LIN {X 0,Y 273.88,Z 288.831,A -85,B 0,C 180,E1 -19129.181,E2 -19129.181} C_VEL
LIN {X 0,Y 275.727,Z 293.143,A -85,B 0,C 180,E1 -19129.643,E2 -19129.643} C_VEL
LIN {X 0,Y 275.975,Z 296.307,A -85,B 0,C 180,E1 -19129.792,E2 -19129.792} C_VEL
LIN {X 0,Y 270.634,Z 402.684,A -85,B 0,C 180,E1 -19132.569,E2 -19132.569} C_VEL
LIN {X 0,Y 269.012,Z 418.51,A -85,B 0,C 180,E1 -19133.244,E2 -19133.244} C_VEL
LIN {X 0,Y 266.872,Z 432.935,A -85,B 0,C 180,E1 -19134.131,E2 -19134.131} C_VEL
LIN {X 0,Y 264.208,Z 447.475,A -85,B 0,C 180,E1 -19135.35,E2 -19135.35} C_VEL
LIN {X 0,Y 261.451,Z 460.406,A -85,B 0,C 180,E1 -19136.749,E2 -19136.749} C_VEL
LIN {X 0,Y 258.282,Z 472.878,A -85,B 0,C 180,E1 -19138.413,E2 -19138.413} C_VEL
LIN {X 0,Y 254.828,Z 485.225,A -85,B 0,C 180,E1 -19140.464,E2 -19140.464} C_VEL
LIN {X 0,Y 251.836,Z 495.611,A -85,B 0,C 180,E1 -19142.584,E2 -19142.584} C_VEL
LIN {X 0,Y 249.001,Z 505.164,A -85,B 0,C 180,E1 -19144.953,E2 -19144.953} C_VEL
LIN {X 0,Y 246.17,Z 514.518,A -85,B 0,C 180,E1 -19147.774,E2 -19147.774} C_VEL
LIN {X 0,Y 243.871,Z 522.241,A -85,B 0,C 180,E1 -19150.646,E2 -19150.646} C_VEL
LIN {X 0,Y 241.943,Z 529.414,A -85,B 0,C 180,E1 -19153.982,E2 -19153.982} C_VEL
LIN {X 0,Y 240.664,Z 535.006,A -85,B 0,C 180,E1 -19157.349,E2 -19157.349} C_VEL
LIN {X 0,Y 240.129,Z 538.242,A -85,B 0,C 180,E1 -19159.887,E2 -19159.887} C_VEL
LIN {X 0,Y 239.909,Z 541.426,A -85,B 0,C 180,E1 -19163.271,E2 -19163.271} C_VEL
LIN {X 0,Y 239.898,Z 543.322,A -85,B 0,C 180,E1 -19166.642,E2 -19166.642} C_VEL
LIN {X 0,Y 239.982,Z 543.802,A -85,B 0,C 180,E1 -19168.322,E2 -19168.322} C_VEL
LIN {X 0,Y 240.016,Z 543.963,A -85,B 0,C 180,E1 -19170.001,E2 -19170.001} C_VEL
LIN {X 0,Y 239.929,Z 543.31,A -85,B 0,C 180,E1 -19173.359,E2 -19173.359} C_VEL
LIN {X 0,Y 239.912,Z 541.395,A -85,B 0,C 180,E1 -19176.73,E2 -19176.73} C_VEL
LIN {X 0,Y 240.135,Z 538.199,A -85,B 0,C 180,E1 -19180.114,E2 -19180.114} C_VEL
LIN {X 0,Y 240.973,Z 533.666,A -85,B 0,C 180,E1 -19183.493,E2 -19183.493} C_VEL
LIN {X 0,Y 242.441,Z 527.505,A -85,B 0,C 180,E1 -19186.939,E2 -19186.939} C_VEL
LIN {X 0,Y 244.457,Z 520.065,A -85,B 0,C 180,E1 -19190.182,E2 -19190.182} C_VEL
LIN {X 0,Y 246.984,Z 511.878,A -85,B 0,C 180,E1 -19193.033,E2 -19193.033} C_VEL
LIN {X 0,Y 249.851,Z 502.062,A -85,B 0,C 180,E1 -19195.827,E2 -19195.827} C_VEL
LIN {X 0,Y 252.851,Z 491.816,A -85,B 0,C 180,E1 -19198.198,E2 -19198.198} C_VEL
LIN {X 0,Y 256.079,Z 480.758,A -85,B 0,C 180,E1 -19200.285,E2 -19200.285} C_VEL
LIN {X 0,Y 259.277,Z 468.756,A -85,B 0,C 180,E1 -19202.138,E2 -19202.138} C_VEL
LIN {X 0,Y 262.224,Z 456.425,A -85,B 0,C 180,E1 -19203.681,E2 -19203.681} C_VEL
LIN {X 0,Y 264.902,Z 443.237,A -85,B 0,C 180,E1 -19205.01,E2 -19205.01} C_VEL
LIN {X 0,Y 267.411,Z 428.644,A -85,B 0,C 180,E1 -19206.135,E2 -19206.135} C_VEL
LIN {X 0,Y 269.485,Z 413.425,A -85,B 0,C 180,E1 -19206.974,E2 -19206.974} C_VEL
LIN {X 0,Y 270.658,Z 400.044,A -85,B 0,C 180,E1 -19207.487,E2 -19207.487} C_VEL
LIN {X 0,Y 275.899,Z 295.964,A -85,B 0,C 180,E1 -19210.187,E2 -19210.187} C_VEL
LIN {X 0,Y 275.389,Z 292.436,A -85,B 0,C 180,E1 -19210.392,E2 -19210.392} C_VEL
LIN {X 0,Y 268.16,Z 276.743,A -85,B 0,C 180,E1 -19212.208,E2 -19212.208} C_VEL
LIN {X 0,Y 260.836,Z 262.769,A -85,B 0,C 180,E1 -19214.133,E2 -19214.133} C_VEL
LIN {X 0,Y 253.192,Z 249.822,A -85,B 0,C 180,E1 -19216.264,E2 -19216.264} C_VEL
LIN {X 0,Y 250.126,Z 244.827,A -85,B 0,C 180,E1 -19217.234,E2 -19217.234} C_VEL
LIN {X 0,Y 247.451,Z 236.819,A -85,B 0,C 180,E1 -19220.737,E2 -19220.737} C_VEL
LIN {X 0,Y 244.929,Z 229.833,A -85,B 0,C 180,E1 -19224.212,E2 -19224.212} C_VEL
LIN {X 0,Y 242.946,Z 224.766,A -85,B 0,C 180,E1 -19227.026,E2 -19227.026} C_VEL
LIN {X 0,Y 241.991,Z 222.06,A -85,B 0,C 180,E1 -19228.726,E2 -19228.726} C_VEL
LIN {X 0,Y 242.005,Z 221.929,A -85,B 0,C 180,E1 -19232.313,E2 -19232.313} C_VEL
LIN {X 0,Y 242.057,Z 221.947,A -85,B 0,C 180,E1 -19236.016,E2 -19236.016} C_VEL
LIN {X 0,Y 242.038,Z 221.955,A -85,B 0,C 180,E1 -19239.608,E2 -19239.608} C_VEL
LIN {X 0,Y 242.163,Z 221.939,A -85,B 0,C 180,E1 -19243.278,E2 -19243.278} C_VEL
LIN {X 0,Y 242.18,Z 221.944,A -85,B 0,C 180,E1 -19248.28,E2 -19248.28} C_VEL
LIN {X 0,Y 242.4,Z 221.912,A -85,B 0,C 180,E1 -19251.665,E2 -19251.665} C_VEL
LIN {X 0,Y 242.255,Z 221.921,A -85,B 0,C 180,E1 -19255.007,E2 -19255.007} C_VEL
LIN {X 0,Y 242.636,Z 221.873,A -85,B 0,C 180,E1 -19258.34,E2 -19258.34} C_VEL
LIN {X 0,Y 242.635,Z 221.883,A -85,B 0,C 180,E1 -19261.66,E2 -19261.66} C_VEL
LIN {X 0,Y 242.429,Z 221.902,A -85,B 0,C 180,E1 -19266.732,E2 -19266.732} C_VEL
LIN {X 0,Y 242.314,Z 221.927,A -85,B 0,C 180,E1 -19270.022,E2 -19270.022} C_VEL
LIN {X 0,Y 242.165,Z 221.935,A -85,B 0,C 180,E1 -19275.141,E2 -19275.141} C_VEL
LIN {X 0,Y 242.079,Z 221.951,A -85,B 0,C 180,E1 -19278.624,E2 -19278.624} C_VEL
LIN {X 0,Y 242.05,Z 221.959,A -85,B 0,C 180,E1 -19282.177,E2 -19282.177} C_VEL
LIN {X 0,Y 242.068,Z 221.955,A -85,B 0,C 180,E1 -19285.838,E2 -19285.838} C_VEL
LIN {X 0,Y 242.008,Z 221.926,A -85,B 0,C 180,E1 -19289.584,E2 -19289.584} C_VEL
LIN {X 0,Y 242.018,Z 222.145,A -85,B 0,C 180,E1 -19293.925,E2 -19293.925} C_VEL
LIN {X 0,Y 244.449,Z 228.742,A -85,B 0,C 180,E1 -19297.871,E2 -19297.871} C_VEL
LIN {X 0,Y 247.454,Z 237.474,A -85,B 0,C 180,E1 -19302.402,E2 -19302.402} C_VEL
LIN {X 0,Y 249.709,Z 244.63,A -85,B 0,C 180,E1 -19305.647,E2 -19305.647} C_VEL
LIN {X 0,Y 256.611,Z 256.13,A -85,B 0,C 180,E1 -19307.687,E2 -19307.687} C_VEL
LIN {X 0,Y 263.672,Z 268.748,A -85,B 0,C 180,E1 -19309.582,E2 -19309.582} C_VEL
LIN {X 0,Y 270.664,Z 282.832,A -85,B 0,C 180,E1 -19311.361,E2 -19311.361} C_VEL
LIN {X 0,Y 274.186,Z 291.049,A -85,B 0,C 180,E1 -19312.241,E2 -19312.241} C_VEL
LIN {X 0,Y 275.36,Z 298.415,A -85,B 0,C 180,E1 -19312.671,E2 -19312.671} C_VEL
LIN {X 0,Y 271.22,Z 391.994,A -85,B 0,C 180,E1 -19314.961,E2 -19314.961} C_VEL
LIN {X 0,Y 269.925,Z 406.095,A -85,B 0,C 180,E1 -19315.564,E2 -19315.564} C_VEL
LIN {X 0,Y 268.066,Z 420.441,A -85,B 0,C 180,E1 -19316.482,E2 -19316.482} C_VEL
LIN {X 0,Y 265.719,Z 433.717,A -85,B 0,C 180,E1 -19317.616,E2 -19317.616} C_VEL
LIN {X 0,Y 263.393,Z 445.05,A -85,B 0,C 180,E1 -19318.856,E2 -19318.856} C_VEL
LIN {X 0,Y 260.577,Z 457.105,A -85,B 0,C 180,E1 -19320.513,E2 -19320.513} C_VEL
LIN {X 0,Y 257.386,Z 468.075,A -85,B 0,C 180,E1 -19322.342,E2 -19322.342} C_VEL
LIN {X 0,Y 254.116,Z 478.916,A -85,B 0,C 180,E1 -19324.616,E2 -19324.616} C_VEL
LIN {X 0,Y 251.056,Z 487.933,A -85,B 0,C 180,E1 -19326.926,E2 -19326.926} C_VEL
LIN {X 0,Y 248.642,Z 495.475,A -85,B 0,C 180,E1 -19329.309,E2 -19329.309} C_VEL
LIN {X 0,Y 246.398,Z 501.761,A -85,B 0,C 180,E1 -19331.714,E2 -19331.714} C_VEL
LIN {X 0,Y 244.462,Z 507.033,A -85,B 0,C 180,E1 -19334.15,E2 -19334.15} C_VEL
LIN {X 0,Y 242.597,Z 512.619,A -85,B 0,C 180,E1 -19337.451,E2 -19337.451} C_VEL
LIN {X 0,Y 241.61,Z 515.871,A -85,B 0,C 180,E1 -19339.948,E2 -19339.948} C_VEL
LIN {X 0,Y 240.71,Z 518.975,A -85,B 0,C 180,E1 -19343.293,E2 -19343.293} C_VEL
LIN {X 0,Y 240.255,Z 520.812,A -85,B 0,C 180,E1 -19346.645,E2 -19346.645} C_VEL
LIN {X 0,Y 240.035,Z 521.438,A -85,B 0,C 180,E1 -19349.999,E2 -19349.999} C_VEL
LIN {X 0,Y 240.238,Z 520.857,A -85,B 0,C 180,E1 -19353.354,E2 -19353.354} C_VEL
LIN {X 0,Y 240.738,Z 518.872,A -85,B 0,C 180,E1 -19356.98,E2 -19356.98} C_VEL
LIN {X 0,Y 241.533,Z 516.012,A -85,B 0,C 180,E1 -19360.054,E2 -19360.054} C_VEL
LIN {X 0,Y 242.97,Z 511.598,A -85,B 0,C 180,E1 -19363.379,E2 -19363.379} C_VEL
LIN {X 0,Y 244.935,Z 505.676,A -85,B 0,C 180,E1 -19366.674,E2 -19366.674} C_VEL
LIN {X 0,Y 247.441,Z 499.096,A -85,B 0,C 180,E1 -19369.495,E2 -19369.495} C_VEL
LIN {X 0,Y 249.647,Z 492.247,A -85,B 0,C 180,E1 -19371.9,E2 -19371.9} C_VEL
LIN {X 0,Y 252.399,Z 484.075,A -85,B 0,C 180,E1 -19374.248,E2 -19374.248} C_VEL
LIN {X 0,Y 255.616,Z 474.289,A -85,B 0,C 180,E1 -19376.536,E2 -19376.536} C_VEL
LIN {X 0,Y 258.816,Z 463.477,A -85,B 0,C 180,E1 -19378.593,E2 -19378.593} C_VEL
LIN {X 0,Y 262.006,Z 451.551,A -85,B 0,C 180,E1 -19380.416,E2 -19380.416} C_VEL
LIN {X 0,Y 264.923,Z 438.291,A -85,B 0,C 180,E1 -19382.043,E2 -19382.043} C_VEL
LIN {X 0,Y 267.579,Z 424.058,A -85,B 0,C 180,E1 -19383.361,E2 -19383.361} C_VEL
LIN {X 0,Y 269.551,Z 410.23,A -85,B 0,C 180,E1 -19384.32,E2 -19384.32} C_VEL
LIN {X 0,Y 271.024,Z 395.948,A -85,B 0,C 180,E1 -19385.009,E2 -19385.009} C_VEL
LIN {X 0,Y 271.986,Z 379.589,A -85,B 0,C 180,E1 -19385.49,E2 -19385.49} C_VEL
LIN {X 0,Y 275.472,Z 298.373,A -85,B 0,C 180,E1 -19387.448,E2 -19387.448} C_VEL
LIN {X 0,Y 274.002,Z 290.224,A -85,B 0,C 180,E1 -19387.955,E2 -19387.955} C_VEL
LIN {X 0,Y 266.603,Z 274.248,A -85,B 0,C 180,E1 -19389.811,E2 -19389.811} C_VEL
LIN {X 0,Y 259.689,Z 261.421,A -85,B 0,C 180,E1 -19391.623,E2 -19391.623} C_VEL
LIN {X 0,Y 254.064,Z 251.882,A -85,B 0,C 180,E1 -19393.18,E2 -19393.18} C_VEL
LIN {X 0,Y 249.679,Z 244.552,A -85,B 0,C 180,E1 -19394.534,E2 -19394.534} C_VEL
LIN {X 0,Y 247.059,Z 236.364,A -85,B 0,C 180,E1 -19398.313,E2 -19398.313} C_VEL
LIN {X 0,Y 244.587,Z 229.079,A -85,B 0,C 180,E1 -19402.12,E2 -19402.12} C_VEL
LIN {X 0,Y 241.997,Z 222.05,A -85,B 0,C 180,E1 -19406.385,E2 -19406.385} C_VEL
LIN {X 0,Y 242.01,Z 221.925,A -85,B 0,C 180,E1 -19410.596,E2 -19410.596} C_VEL
LIN {X 0,Y 242.064,Z 221.953,A -85,B 0,C 180,E1 -19414.182,E2 -19414.182} C_VEL
LIN {X 0,Y 242.06,Z 221.959,A -85,B 0,C 180,E1 -19418.29,E2 -19418.29} C_VEL
LIN {X 0,Y 242.159,Z 221.936,A -85,B 0,C 180,E1 -19423.278,E2 -19423.278} C_VEL
LIN {X 0,Y 242.181,Z 221.93,A -85,B 0,C 180,E1 -19428.279,E2 -19428.279} C_VEL
LIN {X 0,Y 242.423,Z 221.902,A -85,B 0,C 180,E1 -19431.665,E2 -19431.665} C_VEL
LIN {X 0,Y 242.256,Z 221.933,A -85,B 0,C 180,E1 -19435.007,E2 -19435.007} C_VEL
LIN {X 0,Y 242.31,Z 221.914,A -85,B 0,C 180,E1 -19436.135,E2 -19436.135} C_VEL
LIN {X 0,Y 241.756,Z 221.985,A -85,B 0,C 180,E1 -19437.526,E2 -19437.526} C_VEL
LIN {X 0,Y 240.253,Z 222.184,A -85,B 0,C 180,E1 -19438.893,E2 -19438.893} C_VEL
LIN {X 0,Y 235.69,Z 222.76,A -85,B 0,C 180,E1 -19442.594,E2 -19442.594} C_VEL
LIN {X 0,Y 235.295,Z 222.799,A -85,B 0,C 180,E1 -19443.564,E2 -19443.564} C_VEL
LIN {X 0,Y 235.399,Z 222.781,A -85,B 0,C 180,E1 -19446.858,E2 -19446.858} C_VEL
LIN {X 0,Y 235.233,Z 222.796,A -85,B 0,C 180,E1 -19450.326,E2 -19450.326} C_VEL
LIN {X 0,Y 235.108,Z 222.823,A -85,B 0,C 180,E1 -19455.606,E2 -19455.606} C_VEL
LIN {X 0,Y 235.004,Z 222.833,A -85,B 0,C 180,E1 -19459.206,E2 -19459.206} C_VEL
LIN {X 0,Y 234.956,Z 222.841,A -85,B 0,C 180,E1 -19462.883,E2 -19462.883} C_VEL
LIN {X 0,Y 234.964,Z 222.8,A -85,B 0,C 180,E1 -19466.658,E2 -19466.658} C_VEL
LIN {X 0,Y 235.004,Z 223.06,A -85,B 0,C 180,E1 -19468.997,E2 -19468.997} C_VEL
LIN {X 0,Y 237.615,Z 229.785,A -85,B 0,C 180,E1 -19473.265,E2 -19473.265} C_VEL
LIN {X 0,Y 240.196,Z 236.746,A -85,B 0,C 180,E1 -19477.088,E2 -19477.088} C_VEL
LIN {X 0,Y 243.007,Z 244.924,A -85,B 0,C 180,E1 -19480.962,E2 -19480.962} C_VEL
LIN {X 0,Y 250.063,Z 256.334,A -85,B 0,C 180,E1 -19483.218,E2 -19483.218} C_VEL
LIN {X 0,Y 257.579,Z 269.259,A -85,B 0,C 180,E1 -19485.384,E2 -19485.384} C_VEL
LIN {X 0,Y 264.546,Z 282.927,A -85,B 0,C 180,E1 -19487.283,E2 -19487.283} C_VEL
LIN {X 0,Y 270.312,Z 295.808,A -85,B 0,C 180,E1 -19488.803,E2 -19488.803} C_VEL
LIN {X 0,Y 270.263,Z 300.618,A -85,B 0,C 180,E1 -19488.963,E2 -19488.963} C_VEL
LIN {X 0,Y 264.923,Z 402.988,A -85,B 0,C 180,E1 -19491.678,E2 -19491.678} C_VEL
LIN {X 0,Y 263.246,Z 418.621,A -85,B 0,C 180,E1 -19492.361,E2 -19492.361} C_VEL
LIN {X 0,Y 260.937,Z 433.531,A -85,B 0,C 180,E1 -19493.304,E2 -19493.304} C_VEL
LIN {X 0,Y 258.376,Z 447.008,A -85,B 0,C 180,E1 -19494.451,E2 -19494.451} C_VEL
LIN {X 0,Y 255.384,Z 460.492,A -85,B 0,C 180,E1 -19495.936,E2 -19495.936} C_VEL
LIN {X 0,Y 251.851,Z 473.666,A -85,B 0,C 180,E1 -19497.746,E2 -19497.746} C_VEL
LIN {X 0,Y 248.31,Z 485.837,A -85,B 0,C 180,E1 -19499.843,E2 -19499.843} C_VEL
LIN {X 0,Y 244.947,Z 496.914,A -85,B 0,C 180,E1 -19502.21,E2 -19502.21} C_VEL
LIN {X 0,Y 242.041,Z 506.25,A -85,B 0,C 180,E1 -19504.642,E2 -19504.642} C_VEL
LIN {X 0,Y 239.542,Z 514.167,A -85,B 0,C 180,E1 -19507.125,E2 -19507.125} C_VEL
LIN {X 0,Y 237.094,Z 521.895,A -85,B 0,C 180,E1 -19510.07,E2 -19510.07} C_VEL
LIN {X 0,Y 235.004,Z 529.249,A -85,B 0,C 180,E1 -19513.591,E2 -19513.591} C_VEL
LIN {X 0,Y 233.68,Z 534.668,A -85,B 0,C 180,E1 -19516.965,E2 -19516.965} C_VEL
LIN {X 0,Y 233.078,Z 537.905,A -85,B 0,C 180,E1 -19519.578,E2 -19519.578} C_VEL
LIN {X 0,Y 232.807,Z 541.09,A -85,B 0,C 180,E1 -19523.065,E2 -19523.065} C_VEL
LIN {X 0,Y 232.836,Z 542.258,A -85,B 0,C 180,E1 -19524.925,E2 -19524.925} C_VEL
LIN {X 0,Y 232.909,Z 543.471,A -85,B 0,C 180,E1 -19528.272,E2 -19528.272} C_VEL
LIN {X 0,Y 232.945,Z 543.632,A -85,B 0,C 180,E1 -19530.001,E2 -19530.001} C_VEL
LIN {X 0,Y 232.914,Z 543.466,A -85,B 0,C 180,E1 -19531.73,E2 -19531.73} C_VEL
LIN {X 0,Y 232.839,Z 542.177,A -85,B 0,C 180,E1 -19535.196,E2 -19535.196} C_VEL
LIN {X 0,Y 232.892,Z 539.622,A -85,B 0,C 180,E1 -19538.679,E2 -19538.679} C_VEL
LIN {X 0,Y 233.417,Z 535.765,A -85,B 0,C 180,E1 -19542.168,E2 -19542.168} C_VEL
LIN {X 0,Y 234.683,Z 530.518,A -85,B 0,C 180,E1 -19545.636,E2 -19545.636} C_VEL
LIN {X 0,Y 236.508,Z 523.736,A -85,B 0,C 180,E1 -19549.079,E2 -19549.079} C_VEL
LIN {X 0,Y 238.702,Z 516.379,A -85,B 0,C 180,E1 -19552.049,E2 -19552.049} C_VEL
LIN {X 0,Y 241.599,Z 507.498,A -85,B 0,C 180,E1 -19554.948,E2 -19554.948} C_VEL
LIN {X 0,Y 244.335,Z 498.4,A -85,B 0,C 180,E1 -19557.402,E2 -19557.402} C_VEL
LIN {X 0,Y 247.707,Z 487.622,A -85,B 0,C 180,E1 -19559.77,E2 -19559.77} C_VEL
LIN {X 0,Y 251.133,Z 475.805,A -85,B 0,C 180,E1 -19561.885,E2 -19561.885} C_VEL
LIN {X 0,Y 254.835,Z 462.281,A -85,B 0,C 180,E1 -19563.803,E2 -19563.803} C_VEL
LIN {X 0,Y 257.55,Z 450.178,A -85,B 0,C 180,E1 -19565.202,E2 -19565.202} C_VEL
LIN {X 0,Y 260.502,Z 435.325,A -85,B 0,C 180,E1 -19566.528,E2 -19566.528} C_VEL
LIN {X 0,Y 262.819,Z 421.037,A -85,B 0,C 180,E1 -19567.471,E2 -19567.471} C_VEL
LIN {X 0,Y 264.51,Z 406.552,A -85,B 0,C 180,E1 -19568.152,E2 -19568.152} C_VEL
LIN {X 0,Y 265.641,Z 389.193,A -85,B 0,C 180,E1 -19568.685,E2 -19568.685} C_VEL
LIN {X 0,Y 270.327,Z 296.159,A -85,B 0,C 180,E1 -19571.134,E2 -19571.134} C_VEL
LIN {X 0,Y 264.564,Z 283.109,A -85,B 0,C 180,E1 -19572.651,E2 -19572.651} C_VEL
LIN {X 0,Y 257.066,Z 268.28,A -85,B 0,C 180,E1 -19574.699,E2 -19574.699} C_VEL
LIN {X 0,Y 249.079,Z 254.654,A -85,B 0,C 180,E1 -19577.011,E2 -19577.011} C_VEL
LIN {X 0,Y 242.941,Z 244.776,A -85,B 0,C 180,E1 -19579.013,E2 -19579.013} C_VEL
LIN {X 0,Y 239.755,Z 235.444,A -85,B 0,C 180,E1 -19583.495,E2 -19583.495} C_VEL
LIN {X 0,Y 237.542,Z 229.478,A -85,B 0,C 180,E1 -19586.787,E2 -19586.787} C_VEL
LIN {X 0,Y 234.982,Z 222.919,A -85,B 0,C 180,E1 -19591.069,E2 -19591.069} C_VEL
LIN {X 0,Y 234.986,Z 222.811,A -85,B 0,C 180,E1 -19595.247,E2 -19595.247} C_VEL
LIN {X 0,Y 235.011,Z 222.826,A -85,B 0,C 180,E1 -19598.97,E2 -19598.97} C_VEL
LIN {X 0,Y 235.096,Z 222.817,A -85,B 0,C 180,E1 -19603.06,E2 -19603.06} C_VEL
LIN {X 0,Y 235.114,Z 222.823,A -85,B 0,C 180,E1 -19607.922,E2 -19607.922} C_VEL
LIN {X 0,Y 235.331,Z 222.789,A -85,B 0,C 180,E1 -19611.413,E2 -19611.413} C_VEL
LIN {X 0,Y 235.392,Z 222.782,A -85,B 0,C 180,E1 -19613.141,E2 -19613.141} C_VEL
LIN {X 0,Y 235.595,Z 222.75,A -85,B 0,C 180,E1 -19618.291,E2 -19618.291} C_VEL
LIN {X 0,Y 235.595,Z 222.759,A -85,B 0,C 180,E1 -19621.71,E2 -19621.71} C_VEL
LIN {X 0,Y 235.404,Z 222.775,A -85,B 0,C 180,E1 -19626.859,E2 -19626.859} C_VEL
LIN {X 0,Y 235.238,Z 222.805,A -85,B 0,C 180,E1 -19630.327,E2 -19630.327} C_VEL
LIN {X 0,Y 235.113,Z 222.811,A -85,B 0,C 180,E1 -19635.607,E2 -19635.607} C_VEL
LIN {X 0,Y 235.02,Z 222.825,A -85,B 0,C 180,E1 -19639.205,E2 -19639.205} C_VEL
LIN {X 0,Y 234.981,Z 222.832,A -85,B 0,C 180,E1 -19642.881,E2 -19642.881} C_VEL
LIN {X 0,Y 234.969,Z 222.819,A -85,B 0,C 180,E1 -19646.658,E2 -19646.658} C_VEL
LIN {X 0,Y 234.956,Z 222.92,A -85,B 0,C 180,E1 -19651.502,E2 -19651.502} C_VEL
LIN {X 0,Y 237.09,Z 228.579,A -85,B 0,C 180,E1 -19655.313,E2 -19655.313} C_VEL
LIN {X 0,Y 239.421,Z 235.162,A -85,B 0,C 180,E1 -19659.133,E2 -19659.133} C_VEL
LIN {X 0,Y 241.762,Z 242.208,A -85,B 0,C 180,E1 -19662.777,E2 -19662.777} C_VEL
LIN {X 0,Y 242.654,Z 244.905,A -85,B 0,C 180,E1 -19663.945,E2 -19663.945} C_VEL
LIN {X 0,Y 249.443,Z 255.789,A -85,B 0,C 180,E1 -19666.073,E2 -19666.073} C_VEL
LIN {X 0,Y 256.661,Z 268.268,A -85,B 0,C 180,E1 -19668.144,E2 -19668.144} C_VEL
LIN {X 0,Y 263.927,Z 282.513,A -85,B 0,C 180,E1 -19670.107,E2 -19670.107} C_VEL
LIN {X 0,Y 268.911,Z 293.794,A -85,B 0,C 180,E1 -19671.408,E2 -19671.408} C_VEL
LIN {X 0,Y 269.823,Z 299.68,A -85,B 0,C 180,E1 -19671.761,E2 -19671.761} C_VEL
LIN {X 0,Y 265.561,Z 391.742,A -85,B 0,C 180,E1 -19674.042,E2 -19674.042} C_VEL
LIN {X 0,Y 264.238,Z 405.997,A -85,B 0,C 180,E1 -19674.656,E2 -19674.656} C_VEL
LIN {X 0,Y 262.409,Z 419.857,A -85,B 0,C 180,E1 -19675.543,E2 -19675.543} C_VEL
LIN {X 0,Y 260.131,Z 432.429,A -85,B 0,C 180,E1 -19676.6,E2 -19676.6} C_VEL
LIN {X 0,Y 257.576,Z 444.547,A -85,B 0,C 180,E1 -19677.923,E2 -19677.923} C_VEL
LIN {X 0,Y 254.428,Z 457.505,A -85,B 0,C 180,E1 -19679.727,E2 -19679.727} C_VEL
LIN {X 0,Y 251.137,Z 468.453,A -85,B 0,C 180,E1 -19681.592,E2 -19681.592} C_VEL
LIN {X 0,Y 247.718,Z 479.28,A -85,B 0,C 180,E1 -19683.912,E2 -19683.912} C_VEL
LIN {X 0,Y 244.544,Z 488.287,A -85,B 0,C 180,E1 -19686.275,E2 -19686.275} C_VEL
LIN {X 0,Y 242.258,Z 494.869,A -85,B 0,C 180,E1 -19688.38,E2 -19688.38} C_VEL
LIN {X 0,Y 240.465,Z 500.135,A -85,B 0,C 180,E1 -19690.36,E2 -19690.36} C_VEL
LIN {X 0,Y 238.197,Z 505.742,A -85,B 0,C 180,E1 -19692.839,E2 -19692.839} C_VEL
LIN {X 0,Y 236.109,Z 511.738,A -85,B 0,C 180,E1 -19696.224,E2 -19696.224} C_VEL
LIN {X 0,Y 234.61,Z 516.207,A -85,B 0,C 180,E1 -19699.645,E2 -19699.645} C_VEL
LIN {X 0,Y 233.663,Z 519.309,A -85,B 0,C 180,E1 -19703.089,E2 -19703.089} C_VEL
LIN {X 0,Y 233.197,Z 521.144,A -85,B 0,C 180,E1 -19706.544,E2 -19706.544} C_VEL
LIN {X 0,Y 232.963,Z 521.77,A -85,B 0,C 180,E1 -19709.999,E2 -19709.999} C_VEL
LIN {X 0,Y 233.18,Z 521.188,A -85,B 0,C 180,E1 -19713.455,E2 -19713.455} C_VEL
LIN {X 0,Y 233.623,Z 519.401,A -85,B 0,C 180,E1 -19716.91,E2 -19716.91} C_VEL
LIN {X 0,Y 234.549,Z 516.345,A -85,B 0,C 180,E1 -19720.356,E2 -19720.356} C_VEL
LIN {X 0,Y 236.058,Z 511.934,A -85,B 0,C 180,E1 -19723.778,E2 -19723.778} C_VEL
LIN {X 0,Y 238.141,Z 506.015,A -85,B 0,C 180,E1 -19727.164,E2 -19727.164} C_VEL
LIN {X 0,Y 240.755,Z 499.439,A -85,B 0,C 180,E1 -19730.059,E2 -19730.059} C_VEL
LIN {X 0,Y 243.061,Z 492.593,A -85,B 0,C 180,E1 -19732.526,E2 -19732.526} C_VEL
LIN {X 0,Y 245.963,Z 484.428,A -85,B 0,C 180,E1 -19734.926,E2 -19734.926} C_VEL
LIN {X 0,Y 249.29,Z 474.654,A -85,B 0,C 180,E1 -19737.265,E2 -19737.265} C_VEL
LIN {X 0,Y 252.612,Z 463.858,A -85,B 0,C 180,E1 -19739.362,E2 -19739.362} C_VEL
LIN {X 0,Y 255.925,Z 451.956,A -85,B 0,C 180,E1 -19741.219,E2 -19741.219} C_VEL
LIN {X 0,Y 258.535,Z 440.703,A -85,B 0,C 180,E1 -19742.645,E2 -19742.645} C_VEL
LIN {X 0,Y 261.151,Z 427.701,A -85,B 0,C 180,E1 -19743.945,E2 -19743.945} C_VEL
LIN {X 0,Y 263.215,Z 415.003,A -85,B 0,C 180,E1 -19744.916,E2 -19744.916} C_VEL
LIN {X 0,Y 264.904,Z 400.881,A -85,B 0,C 180,E1 -19745.708,E2 -19745.708} C_VEL
LIN {X 0,Y 265.934,Z 387.755,A -85,B 0,C 180,E1 -19746.191,E2 -19746.191} C_VEL
LIN {X 0,Y 269.919,Z 299.435,A -85,B 0,C 180,E1 -19748.368,E2 -19748.368} C_VEL
LIN {X 0,Y 268.84,Z 293.344,A -85,B 0,C 180,E1 -19748.76,E2 -19748.76} C_VEL
LIN {X 0,Y 261.921,Z 278.311,A -85,B 0,C 180,E1 -19750.572,E2 -19750.572} C_VEL
LIN {X 0,Y 255.642,Z 266.39,A -85,B 0,C 180,E1 -19752.291,E2 -19752.291} C_VEL
LIN {X 0,Y 248.662,Z 254.334,A -85,B 0,C 180,E1 -19754.324,E2 -19754.324} C_VEL
LIN {X 0,Y 242.555,Z 244.603,A -85,B 0,C 180,E1 -19756.295,E2 -19756.295} C_VEL
LIN {X 0,Y 239.534,Z 235.445,A -85,B 0,C 180,E1 -19760.889,E2 -19760.889} C_VEL
LIN {X 0,Y 237.189,Z 228.848,A -85,B 0,C 180,E1 -19764.704,E2 -19764.704} C_VEL
LIN {X 0,Y 234.942,Z 222.949,A -85,B 0,C 180,E1 -19768.684,E2 -19768.684} C_VEL
LIN {X 0,Y 234.964,Z 222.818,A -85,B 0,C 180,E1 -19773.342,E2 -19773.342} C_VEL
LIN {X 0,Y 235.026,Z 222.833,A -85,B 0,C 180,E1 -19777.967,E2 -19777.967} C_VEL
LIN {X 0,Y 235.092,Z 222.817,A -85,B 0,C 180,E1 -19783.059,E2 -19783.059} C_VEL
LIN {X 0,Y 235.113,Z 222.81,A -85,B 0,C 180,E1 -19787.922,E2 -19787.922} C_VEL
LIN {X 0,Y 235.372,Z 222.782,A -85,B 0,C 180,E1 -19791.414,E2 -19791.414} C_VEL
LIN {X 0,Y 235.399,Z 222.776,A -85,B 0,C 180,E1 -19793.141,E2 -19793.141} C_VEL
LIN {X 0,Y 235.591,Z 222.759,A -85,B 0,C 180,E1 -19798.29,E2 -19798.29} C_VEL
LIN {X 0,Y 235.591,Z 222.75,A -85,B 0,C 180,E1 -19801.709,E2 -19801.709} C_VEL
LIN {X 0,Y 235.295,Z 222.799,A -85,B 0,C 180,E1 -19803.564,E2 -19803.564} C_VEL
LIN {X 0,Y 234.537,Z 222.885,A -85,B 0,C 180,E1 -19804.993,E2 -19804.993} C_VEL
LIN {X 0,Y 231.678,Z 223.251,A -85,B 0,C 180,E1 -19807.326,E2 -19807.326} C_VEL
LIN {X 0,Y 228.464,Z 223.641,A -85,B 0,C 180,E1 -19810.206,E2 -19810.206} C_VEL
LIN {X 0,Y 228.113,Z 223.683,A -85,B 0,C 180,E1 -19811.202,E2 -19811.202} C_VEL
LIN {X 0,Y 228.053,Z 223.702,A -85,B 0,C 180,E1 -19816.102,E2 -19816.102} C_VEL
LIN {X 0,Y 227.938,Z 223.717,A -85,B 0,C 180,E1 -19819.826,E2 -19819.826} C_VEL
LIN {X 0,Y 227.909,Z 223.714,A -85,B 0,C 180,E1 -19823.633,E2 -19823.633} C_VEL
LIN {X 0,Y 227.987,Z 223.868,A -85,B 0,C 180,E1 -19826.264,E2 -19826.264} C_VEL
LIN {X 0,Y 230.825,Z 231.348,A -85,B 0,C 180,E1 -19831.515,E2 -19831.515} C_VEL
LIN {X 0,Y 233.033,Z 237.095,A -85,B 0,C 180,E1 -19834.961,E2 -19834.961} C_VEL
LIN {X 0,Y 235.587,Z 244.383,A -85,B 0,C 180,E1 -19838.79,E2 -19838.79} C_VEL
LIN {X 0,Y 236.461,Z 246.191,A -85,B 0,C 180,E1 -19839.305,E2 -19839.305} C_VEL
LIN {X 0,Y 240.7,Z 252.685,A -85,B 0,C 180,E1 -19840.753,E2 -19840.753} C_VEL
LIN {X 0,Y 245.793,Z 260.753,A -85,B 0,C 180,E1 -19842.389,E2 -19842.389} C_VEL
LIN {X 0,Y 253.089,Z 273.498,A -85,B 0,C 180,E1 -19844.59,E2 -19844.59} C_VEL
LIN {X 0,Y 259.892,Z 287.035,A -85,B 0,C 180,E1 -19846.531,E2 -19846.531} C_VEL
LIN {X 0,Y 264.884,Z 298.314,A -85,B 0,C 180,E1 -19847.908,E2 -19847.908} C_VEL
LIN {X 0,Y 259.374,Z 402.01,A -85,B 0,C 180,E1 -19850.702,E2 -19850.702} C_VEL
LIN {X 0,Y 257.785,Z 417.191,A -85,B 0,C 180,E1 -19851.356,E2 -19851.356} C_VEL
LIN {X 0,Y 255.492,Z 431.86,A -85,B 0,C 180,E1 -19852.264,E2 -19852.264} C_VEL
LIN {X 0,Y 253,Z 444.644,A -85,B 0,C 180,E1 -19853.329,E2 -19853.329} C_VEL
LIN {X 0,Y 250.004,Z 457.869,A -85,B 0,C 180,E1 -19854.745,E2 -19854.745} C_VEL
LIN {X 0,Y 246.585,Z 470.795,A -85,B 0,C 180,E1 -19856.482,E2 -19856.482} C_VEL
LIN {X 0,Y 243.143,Z 482.355,A -85,B 0,C 180,E1 -19858.407,E2 -19858.407} C_VEL
LIN {X 0,Y 239.733,Z 493.063,A -85,B 0,C 180,E1 -19860.592,E2 -19860.592} C_VEL
LIN {X 0,Y 236.514,Z 502.929,A -85,B 0,C 180,E1 -19863.055,E2 -19863.055} C_VEL
LIN {X 0,Y 233.423,Z 512.559,A -85,B 0,C 180,E1 -19866.018,E2 -19866.018} C_VEL
LIN {X 0,Y 230.647,Z 520.512,A -85,B 0,C 180,E1 -19869.022,E2 -19869.022} C_VEL
LIN {X 0,Y 228.39,Z 527.894,A -85,B 0,C 180,E1 -19872.539,E2 -19872.539} C_VEL
LIN {X 0,Y 227.004,Z 533.042,A -85,B 0,C 180,E1 -19875.661,E2 -19875.661} C_VEL
LIN {X 0,Y 226.042,Z 537.569,A -85,B 0,C 180,E1 -19879.249,E2 -19879.249} C_VEL
LIN {X 0,Y 225.718,Z 540.755,A -85,B 0,C 180,E1 -19882.846,E2 -19882.846} C_VEL
LIN {X 0,Y 225.756,Z 542.033,A -85,B 0,C 180,E1 -19884.993,E2 -19884.993} C_VEL
LIN {X 0,Y 225.814,Z 543.138,A -85,B 0,C 180,E1 -19888.217,E2 -19888.217} C_VEL
LIN {X 0,Y 225.875,Z 543.3,A -85,B 0,C 180,E1 -19890.001,E2 -19890.001} C_VEL
LIN {X 0,Y 225.82,Z 543.133,A -85,B 0,C 180,E1 -19891.784,E2 -19891.784} C_VEL
LIN {X 0,Y 225.739,Z 541.842,A -85,B 0,C 180,E1 -19895.36,E2 -19895.36} C_VEL
LIN {X 0,Y 225.808,Z 539.285,A -85,B 0,C 180,E1 -19898.953,E2 -19898.953} C_VEL
LIN {X 0,Y 226.418,Z 535.426,A -85,B 0,C 180,E1 -19902.55,E2 -19902.55} C_VEL
LIN {X 0,Y 227.785,Z 530.177,A -85,B 0,C 180,E1 -19906.122,E2 -19906.122} C_VEL
LIN {X 0,Y 229.722,Z 523.39,A -85,B 0,C 180,E1 -19909.666,E2 -19909.666} C_VEL
LIN {X 0,Y 232.06,Z 516.029,A -85,B 0,C 180,E1 -19912.715,E2 -19912.715} C_VEL
LIN {X 0,Y 234.669,Z 508.523,A -85,B 0,C 180,E1 -19915.263,E2 -19915.263} C_VEL
LIN {X 0,Y 237.507,Z 499.585,A -85,B 0,C 180,E1 -19917.809,E2 -19917.809} C_VEL
LIN {X 0,Y 240.884,Z 489.217,A -85,B 0,C 180,E1 -19920.218,E2 -19920.218} C_VEL
LIN {X 0,Y 244.421,Z 477.775,A -85,B 0,C 180,E1 -19922.381,E2 -19922.381} C_VEL
LIN {X 0,Y 248.039,Z 465.276,A -85,B 0,C 180,E1 -19924.274,E2 -19924.274} C_VEL
LIN {X 0,Y 251.376,Z 451.476,A -85,B 0,C 180,E1 -19925.953,E2 -19925.953} C_VEL
LIN {X 0,Y 254.402,Z 437.036,A -85,B 0,C 180,E1 -19927.303,E2 -19927.303} C_VEL
LIN {X 0,Y 256.759,Z 423.401,A -85,B 0,C 180,E1 -19928.264,E2 -19928.264} C_VEL
LIN {X 0,Y 258.637,Z 409.025,A -85,B 0,C 180,E1 -19928.993,E2 -19928.993} C_VEL
LIN {X 0,Y 259.823,Z 393.08,A -85,B 0,C 180,E1 -19929.531,E2 -19929.531} C_VEL
LIN {X 0,Y 264.772,Z 298.209,A -85,B 0,C 180,E1 -19932.065,E2 -19932.065} C_VEL
LIN {X 0,Y 257.996,Z 283.166,A -85,B 0,C 180,E1 -19933.938,E2 -19933.938} C_VEL
LIN {X 0,Y 251.46,Z 270.645,A -85,B 0,C 180,E1 -19935.816,E2 -19935.816} C_VEL
LIN {X 0,Y 245.187,Z 259.727,A -85,B 0,C 180,E1 -19937.73,E2 -19937.73} C_VEL
LIN {X 0,Y 238.226,Z 248.837,A -85,B 0,C 180,E1 -19940.003,E2 -19940.003} C_VEL
LIN {X 0,Y 235.712,Z 244.802,A -85,B 0,C 180,E1 -19940.961,E2 -19940.961} C_VEL
LIN {X 0,Y 233.362,Z 238.062,A -85,B 0,C 180,E1 -19944.404,E2 -19944.404} C_VEL
LIN {X 0,Y 231.794,Z 233.623,A -85,B 0,C 180,E1 -19946.924,E2 -19946.924} C_VEL
LIN {X 0,Y 228.925,Z 226.584,A -85,B 0,C 180,E1 -19951.586,E2 -19951.586} C_VEL
LIN {X 0,Y 227.972,Z 223.788,A -85,B 0,C 180,E1 -19953.739,E2 -19953.739} C_VEL
LIN {X 0,Y 227.962,Z 223.703,A -85,B 0,C 180,E1 -19958.287,E2 -19958.287} C_VEL
LIN {X 0,Y 228.035,Z 223.694,A -85,B 0,C 180,E1 -19962.826,E2 -19962.826} C_VEL
LIN {X 0,Y 228.072,Z 223.696,A -85,B 0,C 180,E1 -19967.544,E2 -19967.544} C_VEL
LIN {X 0,Y 228.267,Z 223.666,A -85,B 0,C 180,E1 -19971.145,E2 -19971.145} C_VEL
LIN {X 0,Y 228.339,Z 223.663,A -85,B 0,C 180,E1 -19972.928,E2 -19972.928} C_VEL
LIN {X 0,Y 228.554,Z 223.627,A -85,B 0,C 180,E1 -19978.238,E2 -19978.238} C_VEL
LIN {X 0,Y 228.554,Z 223.635,A -85,B 0,C 180,E1 -19981.762,E2 -19981.762} C_VEL
LIN {X 0,Y 228.355,Z 223.652,A -85,B 0,C 180,E1 -19987.072,E2 -19987.072} C_VEL
LIN {X 0,Y 228.159,Z 223.682,A -85,B 0,C 180,E1 -19990.651,E2 -19990.651} C_VEL
LIN {X 0,Y 228.08,Z 223.699,A -85,B 0,C 180,E1 -19994.271,E2 -19994.271} C_VEL
LIN {X 0,Y 228.007,Z 223.71,A -85,B 0,C 180,E1 -19997.953,E2 -19997.953} C_VEL
LIN {X 0,Y 227.961,Z 223.711,A -85,B 0,C 180,E1 -20002.348,E2 -20002.348} C_VEL
LIN {X 0,Y 227.943,Z 223.694,A -85,B 0,C 180,E1 -20006.602,E2 -20006.602} C_VEL
LIN {X 0,Y 227.919,Z 223.849,A -85,B 0,C 180,E1 -20008.93,E2 -20008.93} C_VEL
LIN {X 0,Y 230.215,Z 229.799,A -85,B 0,C 180,E1 -20013.333,E2 -20013.333} C_VEL
LIN {X 0,Y 232.642,Z 236.409,A -85,B 0,C 180,E1 -20017.503,E2 -20017.503} C_VEL
LIN {X 0,Y 235.349,Z 244.6,A -85,B 0,C 180,E1 -20021.91,E2 -20021.91} C_VEL
LIN {X 0,Y 239.817,Z 251.721,A -85,B 0,C 180,E1 -20023.518,E2 -20023.518} C_VEL
LIN {X 0,Y 245.028,Z 259.919,A -85,B 0,C 180,E1 -20025.184,E2 -20025.184} C_VEL
LIN {X 0,Y 252.712,Z 273.487,A -85,B 0,C 180,E1 -20027.49,E2 -20027.49} C_VEL
LIN {X 0,Y 259.749,Z 287.658,A -85,B 0,C 180,E1 -20029.474,E2 -20029.474} C_VEL
LIN {X 0,Y 263.69,Z 296.593,A -85,B 0,C 180,E1 -20030.543,E2 -20030.543} C_VEL
LIN {X 0,Y 264.353,Z 301.183,A -85,B 0,C 180,E1 -20030.821,E2 -20030.821} C_VEL
LIN {X 0,Y 259.993,Z 391.435,A -85,B 0,C 180,E1 -20033.087,E2 -20033.087} C_VEL
LIN {X 0,Y 258.52,Z 406.666,A -85,B 0,C 180,E1 -20033.752,E2 -20033.752} C_VEL
LIN {X 0,Y 256.605,Z 420.404,A -85,B 0,C 180,E1 -20034.649,E2 -20034.649} C_VEL
LIN {X 0,Y 254.247,Z 432.909,A -85,B 0,C 180,E1 -20035.722,E2 -20035.722} C_VEL
LIN {X 0,Y 251.515,Z 445.399,A -85,B 0,C 180,E1 -20037.12,E2 -20037.12} C_VEL
LIN {X 0,Y 248.322,Z 457.904,A -85,B 0,C 180,E1 -20038.901,E2 -20038.901} C_VEL
LIN {X 0,Y 244.937,Z 468.829,A -85,B 0,C 180,E1 -20040.805,E2 -20040.805} C_VEL
LIN {X 0,Y 241.371,Z 479.643,A -85,B 0,C 180,E1 -20043.172,E2 -20043.172} C_VEL
LIN {X 0,Y 238.076,Z 488.639,A -85,B 0,C 180,E1 -20045.589,E2 -20045.589} C_VEL
LIN {X 0,Y 235.529,Z 495.598,A -85,B 0,C 180,E1 -20047.875,E2 -20047.875} C_VEL
LIN {X 0,Y 233.801,Z 500.478,A -85,B 0,C 180,E1 -20049.776,E2 -20049.776} C_VEL
LIN {X 0,Y 230.804,Z 507.713,A -85,B 0,C 180,E1 -20053.185,E2 -20053.185} C_VEL
LIN {X 0,Y 228.756,Z 513.293,A -85,B 0,C 180,E1 -20056.678,E2 -20056.678} C_VEL
LIN {X 0,Y 227.634,Z 516.542,A -85,B 0,C 180,E1 -20059.324,E2 -20059.324} C_VEL
LIN {X 0,Y 226.591,Z 519.716,A -85,B 0,C 180,E1 -20062.99,E2 -20062.99} C_VEL
LIN {X 0,Y 226.141,Z 521.476,A -85,B 0,C 180,E1 -20066.436,E2 -20066.436} C_VEL
LIN {X 0,Y 225.894,Z 522.101,A -85,B 0,C 180,E1 -20069.999,E2 -20069.999} C_VEL
LIN {X 0,Y 226.101,Z 521.521,A -85,B 0,C 180,E1 -20073.563,E2 -20073.563} C_VEL
LIN {X 0,Y 226.568,Z 519.734,A -85,B 0,C 180,E1 -20077.127,E2 -20077.127} C_VEL
LIN {X 0,Y 227.559,Z 516.678,A -85,B 0,C 180,E1 -20080.678,E2 -20080.678} C_VEL
LIN {X 0,Y 229.164,Z 512.268,A -85,B 0,C 180,E1 -20084.201,E2 -20084.201} C_VEL
LIN {X 0,Y 231.369,Z 506.353,A -85,B 0,C 180,E1 -20087.682,E2 -20087.682} C_VEL
LIN {X 0,Y 234.092,Z 499.782,A -85,B 0,C 180,E1 -20090.655,E2 -20090.655} C_VEL
LIN {X 0,Y 236.502,Z 492.939,A -85,B 0,C 180,E1 -20093.187,E2 -20093.187} C_VEL
LIN {X 0,Y 239.543,Z 484.781,A -85,B 0,C 180,E1 -20095.641,E2 -20095.641} C_VEL
LIN {X 0,Y 243.015,Z 475.018,A -85,B 0,C 180,E1 -20098.03,E2 -20098.03} C_VEL
LIN {X 0,Y 246.457,Z 464.239,A -85,B 0,C 180,E1 -20100.171,E2 -20100.171} C_VEL
LIN {X 0,Y 249.908,Z 452.358,A -85,B 0,C 180,E1 -20102.059,E2 -20102.059} C_VEL
LIN {X 0,Y 252.787,Z 440.33,A -85,B 0,C 180,E1 -20103.607,E2 -20103.607} C_VEL
LIN {X 0,Y 255.323,Z 428.193,A -85,B 0,C 180,E1 -20104.83,E2 -20104.83} C_VEL
LIN {X 0,Y 257.45,Z 415.585,A -85,B 0,C 180,E1 -20105.817,E2 -20105.817} C_VEL
LIN {X 0,Y 259.205,Z 401.626,A -85,B 0,C 180,E1 -20106.618,E2 -20106.618} C_VEL
LIN {X 0,Y 260.37,Z 387.337,A -85,B 0,C 180,E1 -20107.152,E2 -20107.152} C_VEL
LIN {X 0,Y 264.419,Z 300.597,A -85,B 0,C 180,E1 -20109.327,E2 -20109.327} C_VEL
LIN {X 0,Y 263.557,Z 296.08,A -85,B 0,C 180,E1 -20109.643,E2 -20109.643} C_VEL
LIN {X 0,Y 255.962,Z 279.604,A -85,B 0,C 180,E1 -20111.736,E2 -20111.736} C_VEL
LIN {X 0,Y 249.288,Z 267.223,A -85,B 0,C 180,E1 -20113.671,E2 -20113.671} C_VEL
LIN {X 0,Y 243.42,Z 257.343,A -85,B 0,C 180,E1 -20115.481,E2 -20115.481} C_VEL
LIN {X 0,Y 237.951,Z 248.798,A -85,B 0,C 180,E1 -20117.281,E2 -20117.281} C_VEL
LIN {X 0,Y 235.239,Z 244.428,A -85,B 0,C 180,E1 -20118.337,E2 -20118.337} C_VEL
LIN {X 0,Y 232.76,Z 236.815,A -85,B 0,C 180,E1 -20122.445,E2 -20122.445} C_VEL
LIN {X 0,Y 230.324,Z 230.074,A -85,B 0,C 180,E1 -20126.685,E2 -20126.685} C_VEL
LIN {X 0,Y 227.922,Z 223.773,A -85,B 0,C 180,E1 -20131.448,E2 -20131.448} C_VEL
LIN {X 0,Y 227.926,Z 223.717,A -85,B 0,C 180,E1 -20134.425,E2 -20134.425} C_VEL
LIN {X 0,Y 227.987,Z 223.712,A -85,B 0,C 180,E1 -20138.289,E2 -20138.289} C_VEL
LIN {X 0,Y 228.031,Z 223.699,A -85,B 0,C 180,E1 -20142.825,E2 -20142.825} C_VEL
LIN {X 0,Y 228.07,Z 223.689,A -85,B 0,C 180,E1 -20147.543,E2 -20147.543} C_VEL
LIN {X 0,Y 228.301,Z 223.665,A -85,B 0,C 180,E1 -20151.146,E2 -20151.146} C_VEL
LIN {X 0,Y 228.35,Z 223.652,A -85,B 0,C 180,E1 -20152.928,E2 -20152.928} C_VEL
LIN {X 0,Y 228.55,Z 223.635,A -85,B 0,C 180,E1 -20158.238,E2 -20158.238} C_VEL
LIN {X 0,Y 228.55,Z 223.627,A -85,B 0,C 180,E1 -20161.762,E2 -20161.762} C_VEL
LIN {X 0,Y 228.35,Z 223.661,A -85,B 0,C 180,E1 -20167.071,E2 -20167.071} C_VEL
LIN {X 0,Y 228.113,Z 223.683,A -85,B 0,C 180,E1 -20171.202,E2 -20171.202} C_VEL
LIN {X 0,Y 227.385,Z 223.78,A -85,B 0,C 180,E1 -20172.675,E2 -20172.675} C_VEL
LIN {X 0,Y 224.496,Z 224.138,A -85,B 0,C 180,E1 -20175.078,E2 -20175.078} C_VEL
LIN {X 0,Y 222.056,Z 224.44,A -85,B 0,C 180,E1 -20177.038,E2 -20177.038} C_VEL
LIN {X 0,Y 220.986,Z 224.572,A -85,B 0,C 180,E1 -20178.561,E2 -20178.561} C_VEL
LIN {X 0,Y 220.884,Z 224.583,A -85,B 0,C 180,E1 -20179.077,E2 -20179.077} C_VEL
LIN {X 0,Y 220.916,Z 224.837,A -85,B 0,C 180,E1 -20183.194,E2 -20183.194} C_VEL
LIN {X 0,Y 222.397,Z 228.383,A -85,B 0,C 180,E1 -20186.258,E2 -20186.258} C_VEL
LIN {X 0,Y 224.957,Z 235,A -85,B 0,C 180,E1 -20191.03,E2 -20191.03} C_VEL
LIN {X 0,Y 227.278,Z 241.289,A -85,B 0,C 180,E1 -20194.894,E2 -20194.894} C_VEL
LIN {X 0,Y 228.744,Z 245.168,A -85,B 0,C 180,E1 -20196.923,E2 -20196.923} C_VEL
LIN {X 0,Y 236.094,Z 256.285,A -85,B 0,C 180,E1 -20199.671,E2 -20199.671} C_VEL
LIN {X 0,Y 244.328,Z 269.909,A -85,B 0,C 180,E1 -20202.42,E2 -20202.42} C_VEL
LIN {X 0,Y 250.9,Z 282.056,A -85,B 0,C 180,E1 -20204.449,E2 -20204.449} C_VEL
LIN {X 0,Y 257.222,Z 295.49,A -85,B 0,C 180,E1 -20206.315,E2 -20206.315} C_VEL
LIN {X 0,Y 259.413,Z 300.459,A -85,B 0,C 180,E1 -20206.941,E2 -20206.941} C_VEL
LIN {X 0,Y 253.791,Z 402.348,A -85,B 0,C 180,E1 -20209.728,E2 -20209.728} C_VEL
LIN {X 0,Y 252.039,Z 418.09,A -85,B 0,C 180,E1 -20210.434,E2 -20210.434} C_VEL
LIN {X 0,Y 249.664,Z 432.465,A -85,B 0,C 180,E1 -20211.351,E2 -20211.351} C_VEL
LIN {X 0,Y 246.889,Z 446.073,A -85,B 0,C 180,E1 -20212.523,E2 -20212.523} C_VEL
LIN {X 0,Y 243.674,Z 459.602,A -85,B 0,C 180,E1 -20214.046,E2 -20214.046} C_VEL
LIN {X 0,Y 239.897,Z 472.876,A -85,B 0,C 180,E1 -20215.926,E2 -20215.926} C_VEL
LIN {X 0,Y 236.442,Z 484.098,A -85,B 0,C 180,E1 -20217.907,E2 -20217.907} C_VEL
LIN {X 0,Y 232.927,Z 494.504,A -85,B 0,C 180,E1 -20220.144,E2 -20220.144} C_VEL
LIN {X 0,Y 229.619,Z 504.084,A -85,B 0,C 180,E1 -20222.672,E2 -20222.672} C_VEL
LIN {X 0,Y 226.423,Z 513.467,A -85,B 0,C 180,E1 -20225.716,E2 -20225.716} C_VEL
LIN {X 0,Y 223.593,Z 521.201,A -85,B 0,C 180,E1 -20228.811,E2 -20228.811} C_VEL
LIN {X 0,Y 221.387,Z 528.028,A -85,B 0,C 180,E1 -20232.242,E2 -20232.242} C_VEL
LIN {X 0,Y 219.727,Z 533.99,A -85,B 0,C 180,E1 -20236.121,E2 -20236.121} C_VEL
LIN {X 0,Y 219.001,Z 537.232,A -85,B 0,C 180,E1 -20238.899,E2 -20238.899} C_VEL
LIN {X 0,Y 218.622,Z 540.42,A -85,B 0,C 180,E1 -20242.613,E2 -20242.613} C_VEL
LIN {X 0,Y 218.67,Z 541.816,A -85,B 0,C 180,E1 -20245.088,E2 -20245.088} C_VEL
LIN {X 0,Y 218.722,Z 542.805,A -85,B 0,C 180,E1 -20248.159,E2 -20248.159} C_VEL
LIN {X 0,Y 218.805,Z 542.968,A -85,B 0,C 180,E1 -20250.001,E2 -20250.001} C_VEL
LIN {X 0,Y 218.643,Z 542.309,A -85,B 0,C 180,E1 -20253.687,E2 -20253.687} C_VEL
LIN {X 0,Y 218.628,Z 540.387,A -85,B 0,C 180,E1 -20257.388,E2 -20257.388} C_VEL
LIN {X 0,Y 219.009,Z 537.185,A -85,B 0,C 180,E1 -20261.102,E2 -20261.102} C_VEL
LIN {X 0,Y 220.081,Z 532.644,A -85,B 0,C 180,E1 -20264.802,E2 -20264.802} C_VEL
LIN {X 0,Y 221.806,Z 526.64,A -85,B 0,C 180,E1 -20268.473,E2 -20268.473} C_VEL
LIN {X 0,Y 224.324,Z 519.02,A -85,B 0,C 180,E1 -20272.084,E2 -20272.084} C_VEL
LIN {X 0,Y 227.279,Z 510.814,A -85,B 0,C 180,E1 -20275.163,E2 -20275.163} C_VEL
LIN {X 0,Y 230.516,Z 501.197,A -85,B 0,C 180,E1 -20278.102,E2 -20278.102} C_VEL
LIN {X 0,Y 234.084,Z 490.688,A -85,B 0,C 180,E1 -20280.691,E2 -20280.691} C_VEL
LIN {X 0,Y 237.711,Z 479.575,A -85,B 0,C 180,E1 -20282.906,E2 -20282.906} C_VEL
LIN {X 0,Y 241.406,Z 467.505,A -85,B 0,C 180,E1 -20284.844,E2 -20284.844} C_VEL
LIN {X 0,Y 244.69,Z 454.809,A -85,B 0,C 180,E1 -20286.504,E2 -20286.504} C_VEL
LIN {X 0,Y 247.702,Z 441.714,A -85,B 0,C 180,E1 -20287.848,E2 -20287.848} C_VEL
LIN {X 0,Y 250.264,Z 428.152,A -85,B 0,C 180,E1 -20288.928,E2 -20288.928} C_VEL
LIN {X 0,Y 252.529,Z 412.966,A -85,B 0,C 180,E1 -20289.799,E2 -20289.799} C_VEL
LIN {X 0,Y 253.815,Z 399.625,A -85,B 0,C 180,E1 -20290.334,E2 -20290.334} C_VEL
LIN {X 0,Y 259.328,Z 301.568,A -85,B 0,C 180,E1 -20292.978,E2 -20292.978} C_VEL
LIN {X 0,Y 259.071,Z 299.829,A -85,B 0,C 180,E1 -20293.094,E2 -20293.094} C_VEL
LIN {X 0,Y 251.839,Z 284.034,A -85,B 0,C 180,E1 -20295.199,E2 -20295.199} C_VEL
LIN {X 0,Y 245.179,Z 271.469,A -85,B 0,C 180,E1 -20297.235,E2 -20297.235} C_VEL
LIN {X 0,Y 238.063,Z 259.442,A -85,B 0,C 180,E1 -20299.567,E2 -20299.567} C_VEL
LIN {X 0,Y 231.649,Z 249.593,A -85,B 0,C 180,E1 -20301.841,E2 -20301.841} C_VEL
LIN {X 0,Y 228.512,Z 244.713,A -85,B 0,C 180,E1 -20303.146,E2 -20303.146} C_VEL
LIN {X 0,Y 226.051,Z 237.737,A -85,B 0,C 180,E1 -20307.081,E2 -20307.081} C_VEL
LIN {X 0,Y 223.817,Z 232.041,A -85,B 0,C 180,E1 -20310.877,E2 -20310.877} C_VEL
LIN {X 0,Y 222.349,Z 228.186,A -85,B 0,C 180,E1 -20313.736,E2 -20313.736} C_VEL
LIN {X 0,Y 220.877,Z 224.668,A -85,B 0,C 180,E1 -20316.924,E2 -20316.924} C_VEL
LIN {X 0,Y 220.922,Z 224.581,A -85,B 0,C 180,E1 -20321.451,E2 -20321.451} C_VEL
LIN {X 0,Y 220.996,Z 224.572,A -85,B 0,C 180,E1 -20325.262,E2 -20325.262} C_VEL
LIN {X 0,Y 221.205,Z 224.543,A -85,B 0,C 180,E1 -20330.86,E2 -20330.86} C_VEL
LIN {X 0,Y 221.272,Z 224.546,A -85,B 0,C 180,E1 -20332.701,E2 -20332.701} C_VEL
LIN {X 0,Y 221.512,Z 224.504,A -85,B 0,C 180,E1 -20338.182,E2 -20338.182} C_VEL
LIN {X 0,Y 221.512,Z 224.511,A -85,B 0,C 180,E1 -20341.818,E2 -20341.818} C_VEL
LIN {X 0,Y 221.29,Z 224.531,A -85,B 0,C 180,E1 -20347.299,E2 -20347.299} C_VEL
LIN {X 0,Y 221.108,Z 224.557,A -85,B 0,C 180,E1 -20350.995,E2 -20350.995} C_VEL
LIN {X 0,Y 221.017,Z 224.567,A -85,B 0,C 180,E1 -20356.63,E2 -20356.63} C_VEL
LIN {X 0,Y 220.91,Z 224.581,A -85,B 0,C 180,E1 -20360.485,E2 -20360.485} C_VEL
LIN {X 0,Y 220.874,Z 224.588,A -85,B 0,C 180,E1 -20364.435,E2 -20364.435} C_VEL
LIN {X 0,Y 220.926,Z 224.818,A -85,B 0,C 180,E1 -20365.939,E2 -20365.939} C_VEL
LIN {X 0,Y 223.491,Z 231.356,A -85,B 0,C 180,E1 -20371.366,E2 -20371.366} C_VEL
LIN {X 0,Y 225.473,Z 236.65,A -85,B 0,C 180,E1 -20375.04,E2 -20375.04} C_VEL
LIN {X 0,Y 227.756,Z 243.446,A -85,B 0,C 180,E1 -20379.161,E2 -20379.161} C_VEL
LIN {X 0,Y 228.46,Z 245.199,A -85,B 0,C 180,E1 -20379.916,E2 -20379.916} C_VEL
LIN {X 0,Y 233.128,Z 252.226,A -85,B 0,C 180,E1 -20381.683,E2 -20381.683} C_VEL
LIN {X 0,Y 236.676,Z 257.722,A -85,B 0,C 180,E1 -20382.932,E2 -20382.932} C_VEL
LIN {X 0,Y 241.69,Z 265.896,A -85,B 0,C 180,E1 -20384.6,E2 -20384.6} C_VEL
LIN {X 0,Y 248.392,Z 277.905,A -85,B 0,C 180,E1 -20386.693,E2 -20386.693} C_VEL
LIN {X 0,Y 255.258,Z 292.004,A -85,B 0,C 180,E1 -20388.718,E2 -20388.718} C_VEL
LIN {X 0,Y 258.653,Z 299.859,A -85,B 0,C 180,E1 -20389.685,E2 -20389.685} C_VEL
LIN {X 0,Y 258.87,Z 303.628,A -85,B 0,C 180,E1 -20389.859,E2 -20389.859} C_VEL
LIN {X 0,Y 254.354,Z 392.545,A -85,B 0,C 180,E1 -20392.132,E2 -20392.132} C_VEL
LIN {X 0,Y 252.859,Z 407.337,A -85,B 0,C 180,E1 -20392.805,E2 -20392.805} C_VEL
LIN {X 0,Y 250.886,Z 420.949,A -85,B 0,C 180,E1 -20393.717,E2 -20393.717} C_VEL
LIN {X 0,Y 248.442,Z 433.383,A -85,B 0,C 180,E1 -20394.804,E2 -20394.804} C_VEL
LIN {X 0,Y 245.51,Z 446.212,A -85,B 0,C 180,E1 -20396.276,E2 -20396.276} C_VEL
LIN {X 0,Y 242.288,Z 458.302,A -85,B 0,C 180,E1 -20398.037,E2 -20398.037} C_VEL
LIN {X 0,Y 238.775,Z 469.206,A -85,B 0,C 180,E1 -20399.975,E2 -20399.975} C_VEL
LIN {X 0,Y 235.07,Z 480.005,A -85,B 0,C 180,E1 -20402.392,E2 -20402.392} C_VEL
LIN {X 0,Y 231.632,Z 488.991,A -85,B 0,C 180,E1 -20404.863,E2 -20404.863} C_VEL
LIN {X 0,Y 228.824,Z 496.318,A -85,B 0,C 180,E1 -20407.338,E2 -20407.338} C_VEL
LIN {X 0,Y 226.279,Z 502.792,A -85,B 0,C 180,E1 -20410.022,E2 -20410.022} C_VEL
LIN {X 0,Y 224.003,Z 508.052,A -85,B 0,C 180,E1 -20412.659,E2 -20412.659} C_VEL
LIN {X 0,Y 221.835,Z 513.63,A -85,B 0,C 180,E1 -20416.254,E2 -20416.254} C_VEL
LIN {X 0,Y 220.652,Z 516.877,A -85,B 0,C 180,E1 -20418.982,E2 -20418.982} C_VEL
LIN {X 0,Y 219.589,Z 519.976,A -85,B 0,C 180,E1 -20422.644,E2 -20422.644} C_VEL
LIN {X 0,Y 219.063,Z 521.809,A -85,B 0,C 180,E1 -20426.321,E2 -20426.321} C_VEL
LIN {X 0,Y 218.826,Z 522.433,A -85,B 0,C 180,E1 -20429.999,E2 -20429.999} C_VEL
LIN {X 0,Y 219.025,Z 521.853,A -85,B 0,C 180,E1 -20433.679,E2 -20433.679} C_VEL
LIN {X 0,Y 219.526,Z 520.066,A -85,B 0,C 180,E1 -20437.357,E2 -20437.357} C_VEL
LIN {X 0,Y 220.571,Z 517.012,A -85,B 0,C 180,E1 -20441.021,E2 -20441.021} C_VEL
LIN {X 0,Y 222.265,Z 512.604,A -85,B 0,C 180,E1 -20444.652,E2 -20444.652} C_VEL
LIN {X 0,Y 224.622,Z 506.691,A -85,B 0,C 180,E1 -20448.232,E2 -20448.232} C_VEL
LIN {X 0,Y 227.443,Z 500.125,A -85,B 0,C 180,E1 -20451.288,E2 -20451.288} C_VEL
LIN {X 0,Y 230.496,Z 492.042,A -85,B 0,C 180,E1 -20454.306,E2 -20454.306} C_VEL
LIN {X 0,Y 233.806,Z 483.666,A -85,B 0,C 180,E1 -20456.799,E2 -20456.799} C_VEL
LIN {X 0,Y 237.385,Z 473.614,A -85,B 0,C 180,E1 -20459.241,E2 -20459.241} C_VEL
LIN {X 0,Y 241.063,Z 462.462,A -85,B 0,C 180,E1 -20461.407,E2 -20461.407} C_VEL
LIN {X 0,Y 244.306,Z 451.476,A -85,B 0,C 180,E1 -20463.131,E2 -20463.131} C_VEL
LIN {X 0,Y 247.176,Z 439.626,A -85,B 0,C 180,E1 -20464.656,E2 -20464.656} C_VEL
LIN {X 0,Y 249.941,Z 426.704,A -85,B 0,C 180,E1 -20465.941,E2 -20465.941} C_VEL
LIN {X 0,Y 252.355,Z 412.171,A -85,B 0,C 180,E1 -20467.03,E2 -20467.03} C_VEL
LIN {X 0,Y 254.077,Z 397.447,A -85,B 0,C 180,E1 -20467.795,E2 -20467.795} C_VEL
LIN {X 0,Y 255.151,Z 381.71,A -85,B 0,C 180,E1 -20468.296,E2 -20468.296} C_VEL
LIN {X 0,Y 259.038,Z 301.924,A -85,B 0,C 180,E1 -20470.314,E2 -20470.314} C_VEL
LIN {X 0,Y 258.505,Z 299.32,A -85,B 0,C 180,E1 -20470.511,E2 -20470.511} C_VEL
LIN {X 0,Y 251.787,Z 284.403,A -85,B 0,C 180,E1 -20472.453,E2 -20472.453} C_VEL
LIN {X 0,Y 245.337,Z 272.23,A -85,B 0,C 180,E1 -20474.403,E2 -20474.403} C_VEL
LIN {X 0,Y 238.253,Z 259.977,A -85,B 0,C 180,E1 -20476.713,E2 -20476.713} C_VEL
LIN {X 0,Y 231.223,Z 249.34,A -85,B 0,C 180,E1 -20479.192,E2 -20479.192} C_VEL
LIN {X 0,Y 228.08,Z 244.408,A -85,B 0,C 180,E1 -20480.52,E2 -20480.52} C_VEL
LIN {X 0,Y 226.133,Z 238.624,A -85,B 0,C 180,E1 -20483.904,E2 -20483.904} C_VEL
LIN {X 0,Y 224.579,Z 234.225,A -85,B 0,C 180,E1 -20486.794,E2 -20486.794} C_VEL
LIN {X 0,Y 222.093,Z 227.803,A -85,B 0,C 180,E1 -20491.662,E2 -20491.662} C_VEL
LIN {X 0,Y 220.882,Z 224.659,A -85,B 0,C 180,E1 -20494.561,E2 -20494.561} C_VEL
LIN {X 0,Y 220.92,Z 224.585,A -85,B 0,C 180,E1 -20497.558,E2 -20497.558} C_VEL
LIN {X 0,Y 220.981,Z 224.579,A -85,B 0,C 180,E1 -20502.57,E2 -20502.57} C_VEL
LIN {X 0,Y 221.008,Z 224.571,A -85,B 0,C 180,E1 -20507.138,E2 -20507.138} C_VEL
LIN {X 0,Y 221.232,Z 224.548,A -85,B 0,C 180,E1 -20510.86,E2 -20510.86} C_VEL
LIN {X 0,Y 221.285,Z 224.531,A -85,B 0,C 180,E1 -20512.701,E2 -20512.701} C_VEL
LIN {X 0,Y 221.508,Z 224.511,A -85,B 0,C 180,E1 -20518.181,E2 -20518.181} C_VEL
LIN {X 0,Y 221.508,Z 224.504,A -85,B 0,C 180,E1 -20521.818,E2 -20521.818} C_VEL
LIN {X 0,Y 221.301,Z 224.542,A -85,B 0,C 180,E1 -20527.298,E2 -20527.298} C_VEL
LIN {X 0,Y 221.09,Z 224.56,A -85,B 0,C 180,E1 -20531.157,E2 -20531.157} C_VEL
LIN {X 0,Y 221.012,Z 224.572,A -85,B 0,C 180,E1 -20536.63,E2 -20536.63} C_VEL
LIN {X 0,Y 220.884,Z 224.583,A -85,B 0,C 180,E1 -20539.077,E2 -20539.077} C_VEL
LIN {X 0,Y 220.39,Z 225.162,A -85,B 0,C 180,E1 -20540.593,E2 -20540.593} C_VEL
LIN {X 0,Y 219.35,Z 226.626,A -85,B 0,C 180,E1 -20542.066,E2 -20542.066} C_VEL
LIN {X 0,Y 217.234,Z 230.936,A -85,B 0,C 180,E1 -20544.961,E2 -20544.961} C_VEL
LIN {X 0,Y 217.112,Z 233.877,A -85,B 0,C 180,E1 -20546.928,E2 -20546.928} C_VEL
LIN {X 0,Y 219.256,Z 239.184,A -85,B 0,C 180,E1 -20550.854,E2 -20550.854} C_VEL
LIN {X 0,Y 221.425,Z 245.024,A -85,B 0,C 180,E1 -20554.444,E2 -20554.444} C_VEL
LIN {X 0,Y 226.219,Z 252.09,A -85,B 0,C 180,E1 -20556.501,E2 -20556.501} C_VEL
LIN {X 0,Y 230.445,Z 258.413,A -85,B 0,C 180,E1 -20558.139,E2 -20558.139} C_VEL
LIN {X 0,Y 235.615,Z 266.734,A -85,B 0,C 180,E1 -20560.02,E2 -20560.02} C_VEL
LIN {X 0,Y 242.699,Z 279.026,A -85,B 0,C 180,E1 -20562.409,E2 -20562.409} C_VEL
LIN {X 0,Y 249.607,Z 292.744,A -85,B 0,C 180,E1 -20564.595,E2 -20564.595} C_VEL
LIN {X 0,Y 254.068,Z 302.874,A -85,B 0,C 180,E1 -20565.953,E2 -20565.953} C_VEL
LIN {X 0,Y 248.392,Z 401.315,A -85,B 0,C 180,E1 -20568.664,E2 -20568.664} C_VEL
LIN {X 0,Y 246.69,Z 416.638,A -85,B 0,C 180,E1 -20569.332,E2 -20569.332} C_VEL
LIN {X 0,Y 244.16,Z 431.934,A -85,B 0,C 180,E1 -20570.31,E2 -20570.31} C_VEL
LIN {X 0,Y 241.287,Z 445.606,A -85,B 0,C 180,E1 -20571.496,E2 -20571.496} C_VEL
LIN {X 0,Y 237.926,Z 459.153,A -85,B 0,C 180,E1 -20573.031,E2 -20573.031} C_VEL
LIN {X 0,Y 234.03,Z 472.482,A -85,B 0,C 180,E1 -20574.949,E2 -20574.949} C_VEL
LIN {X 0,Y 230.359,Z 483.719,A -85,B 0,C 180,E1 -20576.953,E2 -20576.953} C_VEL
LIN {X 0,Y 226.714,Z 494.134,A -85,B 0,C 180,E1 -20579.238,E2 -20579.238} C_VEL
LIN {X 0,Y 222.872,Z 504.841,A -85,B 0,C 180,E1 -20582.155,E2 -20582.155} C_VEL
LIN {X 0,Y 219.424,Z 514.316,A -85,B 0,C 180,E1 -20585.395,E2 -20585.395} C_VEL
LIN {X 0,Y 216.916,Z 520.856,A -85,B 0,C 180,E1 -20588.125,E2 -20588.125} C_VEL
LIN {X 0,Y 214.416,Z 528.122,A -85,B 0,C 180,E1 -20591.904,E2 -20591.904} C_VEL
LIN {X 0,Y 212.759,Z 533.651,A -85,B 0,C 180,E1 -20595.657,E2 -20595.657} C_VEL
LIN {X 0,Y 211.956,Z 536.895,A -85,B 0,C 180,E1 -20598.525,E2 -20598.525} C_VEL
LIN {X 0,Y 211.552,Z 540.086,A -85,B 0,C 180,E1 -20602.365,E2 -20602.365} C_VEL
LIN {X 0,Y 211.563,Z 541.63,A -85,B 0,C 180,E1 -20605.258,E2 -20605.258} C_VEL
LIN {X 0,Y 211.632,Z 542.472,A -85,B 0,C 180,E1 -20608.098,E2 -20608.098} C_VEL
LIN {X 0,Y 211.737,Z 542.637,A -85,B 0,C 180,E1 -20610.001,E2 -20610.001} C_VEL
LIN {X 0,Y 211.558,Z 541.976,A -85,B 0,C 180,E1 -20613.81,E2 -20613.81} C_VEL
LIN {X 0,Y 211.559,Z 540.051,A -85,B 0,C 180,E1 -20617.637,E2 -20617.637} C_VEL
LIN {X 0,Y 211.965,Z 536.846,A -85,B 0,C 180,E1 -20621.475,E2 -20621.475} C_VEL
LIN {X 0,Y 213.134,Z 532.302,A -85,B 0,C 180,E1 -20625.296,E2 -20625.296} C_VEL
LIN {X 0,Y 214.994,Z 526.295,A -85,B 0,C 180,E1 -20629.081,E2 -20629.081} C_VEL
LIN {X 0,Y 217.671,Z 518.672,A -85,B 0,C 180,E1 -20632.796,E2 -20632.796} C_VEL
LIN {X 0,Y 220.791,Z 510.46,A -85,B 0,C 180,E1 -20635.956,E2 -20635.956} C_VEL
LIN {X 0,Y 223.765,Z 502.045,A -85,B 0,C 180,E1 -20638.619,E2 -20638.619} C_VEL
LIN {X 0,Y 227.319,Z 492.124,A -85,B 0,C 180,E1 -20641.189,E2 -20641.189} C_VEL
LIN {X 0,Y 231.37,Z 480.265,A -85,B 0,C 180,E1 -20643.666,E2 -20643.666} C_VEL
LIN {X 0,Y 235.186,Z 468.393,A -85,B 0,C 180,E1 -20645.642,E2 -20645.642} C_VEL
LIN {X 0,Y 238.84,Z 454.901,A -85,B 0,C 180,E1 -20647.459,E2 -20647.459} C_VEL
LIN {X 0,Y 242.119,Z 441.207,A -85,B 0,C 180,E1 -20648.882,E2 -20648.882} C_VEL
LIN {X 0,Y 244.761,Z 427.555,A -85,B 0,C 180,E1 -20649.976,E2 -20649.976} C_VEL
LIN {X 0,Y 247.118,Z 412.211,A -85,B 0,C 180,E1 -20650.853,E2 -20650.853} C_VEL
LIN {X 0,Y 248.417,Z 398.502,A -85,B 0,C 180,E1 -20651.399,E2 -20651.399} C_VEL
LIN {X 0,Y 253.944,Z 302.781,A -85,B 0,C 180,E1 -20654.018,E2 -20654.018} C_VEL
LIN {X 0,Y 247.221,Z 287.971,A -85,B 0,C 180,E1 -20656.072,E2 -20656.072} C_VEL
LIN {X 0,Y 241.234,Z 276.4,A -85,B 0,C 180,E1 -20657.993,E2 -20657.993} C_VEL
LIN {X 0,Y 234.123,Z 264.234,A -85,B 0,C 180,E1 -20660.428,E2 -20660.428} C_VEL
LIN {X 0,Y 228.01,Z 254.723,A -85,B 0,C 180,E1 -20662.699,E2 -20662.699} C_VEL
LIN {X 0,Y 224.098,Z 249.044,A -85,B 0,C 180,E1 -20664.261,E2 -20664.261} C_VEL
LIN {X 0,Y 221.261,Z 244.675,A -85,B 0,C 180,E1 -20665.598,E2 -20665.598} C_VEL
LIN {X 0,Y 219.223,Z 238.985,A -85,B 0,C 180,E1 -20669.141,E2 -20669.141} C_VEL
LIN {X 0,Y 216.687,Z 232.403,A -85,B 0,C 180,E1 -20674.033,E2 -20674.033} C_VEL
LIN {X 0,Y 215.325,Z 229.076,A -85,B 0,C 180,E1 -20676.942,E2 -20676.942} C_VEL
LIN {X 0,Y 213.871,Z 225.604,A -85,B 0,C 180,E1 -20680.567,E2 -20680.567} C_VEL
LIN {X 0,Y 213.934,Z 225.455,A -85,B 0,C 180,E1 -20684.763,E2 -20684.763} C_VEL
LIN {X 0,Y 214.142,Z 225.422,A -85,B 0,C 180,E1 -20690.556,E2 -20690.556} C_VEL
LIN {X 0,Y 214.208,Z 225.428,A -85,B 0,C 180,E1 -20692.459,E2 -20692.459} C_VEL
LIN {X 0,Y 214.445,Z 225.384,A -85,B 0,C 180,E1 -20698.122,E2 -20698.122} C_VEL
LIN {X 0,Y 214.546,Z 225.375,A -85,B 0,C 180,E1 -20700,E2 -20700} C_VEL
LIN {X 0,Y 214.445,Z 225.39,A -85,B 0,C 180,E1 -20701.878,E2 -20701.878} C_VEL
LIN {X 0,Y 214.228,Z 225.41,A -85,B 0,C 180,E1 -20707.541,E2 -20707.541} C_VEL
LIN {X 0,Y 214.025,Z 225.437,A -85,B 0,C 180,E1 -20711.363,E2 -20711.363} C_VEL
LIN {X 0,Y 213.941,Z 225.449,A -85,B 0,C 180,E1 -20715.237,E2 -20715.237} C_VEL
LIN {X 0,Y 213.877,Z 225.458,A -85,B 0,C 180,E1 -20719.184,E2 -20719.184} C_VEL
LIN {X 0,Y 213.898,Z 225.704,A -85,B 0,C 180,E1 -20722.201,E2 -20722.201} C_VEL
LIN {X 0,Y 215.403,Z 229.538,A -85,B 0,C 180,E1 -20726.134,E2 -20726.134} C_VEL
LIN {X 0,Y 217.719,Z 235.364,A -85,B 0,C 180,E1 -20731.097,E2 -20731.097} C_VEL
LIN {X 0,Y 219.785,Z 241.068,A -85,B 0,C 180,E1 -20735.141,E2 -20735.141} C_VEL
LIN {X 0,Y 221.118,Z 244.808,A -85,B 0,C 180,E1 -20737.407,E2 -20737.407} C_VEL
LIN {X 0,Y 224.563,Z 249.855,A -85,B 0,C 180,E1 -20738.904,E2 -20738.904} C_VEL
LIN {X 0,Y 229.513,Z 257.298,A -85,B 0,C 180,E1 -20740.844,E2 -20740.844} C_VEL
LIN {X 0,Y 235.443,Z 266.789,A -85,B 0,C 180,E1 -20742.992,E2 -20742.992} C_VEL
LIN {X 0,Y 241.945,Z 278.174,A -85,B 0,C 180,E1 -20745.17,E2 -20745.17} C_VEL
LIN {X 0,Y 249.167,Z 292.69,A -85,B 0,C 180,E1 -20747.437,E2 -20747.437} C_VEL
LIN {X 0,Y 253.561,Z 302.708,A -85,B 0,C 180,E1 -20748.753,E2 -20748.753} C_VEL
LIN {X 0,Y 249.433,Z 385.011,A -85,B 0,C 180,E1 -20750.876,E2 -20750.876} C_VEL
LIN {X 0,Y 248.369,Z 399.171,A -85,B 0,C 180,E1 -20751.373,E2 -20751.373} C_VEL
LIN {X 0,Y 246.639,Z 412.601,A -85,B 0,C 180,E1 -20752.09,E2 -20752.09} C_VEL
LIN {X 0,Y 244.196,Z 427.039,A -85,B 0,C 180,E1 -20753.202,E2 -20753.202} C_VEL
LIN {X 0,Y 241.182,Z 440.266,A -85,B 0,C 180,E1 -20754.534,E2 -20754.534} C_VEL
LIN {X 0,Y 238.13,Z 452.429,A -85,B 0,C 180,E1 -20756.147,E2 -20756.147} C_VEL
LIN {X 0,Y 234.418,Z 464.391,A -85,B 0,C 180,E1 -20758.102,E2 -20758.102} C_VEL
LIN {X 0,Y 230.672,Z 475.234,A -85,B 0,C 180,E1 -20760.324,E2 -20760.324} C_VEL
LIN {X 0,Y 226.98,Z 485.055,A -85,B 0,C 180,E1 -20762.825,E2 -20762.825} C_VEL
LIN {X 0,Y 223.609,Z 493.272,A -85,B 0,C 180,E1 -20765.389,E2 -20765.389} C_VEL
LIN {X 0,Y 220.553,Z 501.162,A -85,B 0,C 180,E1 -20768.503,E2 -20768.503} C_VEL
LIN {X 0,Y 217.232,Z 508.391,A -85,B 0,C 180,E1 -20772.1,E2 -20772.1} C_VEL
LIN {X 0,Y 214.925,Z 513.967,A -85,B 0,C 180,E1 -20775.803,E2 -20775.803} C_VEL
LIN {X 0,Y 213.673,Z 517.212,A -85,B 0,C 180,E1 -20778.618,E2 -20778.618} C_VEL
LIN {X 0,Y 212.556,Z 520.309,A -85,B 0,C 180,E1 -20782.399,E2 -20782.399} C_VEL
LIN {X 0,Y 211.989,Z 522.142,A -85,B 0,C 180,E1 -20786.198,E2 -20786.198} C_VEL
LIN {X 0,Y 211.76,Z 522.765,A -85,B 0,C 180,E1 -20789.999,E2 -20789.999} C_VEL
LIN {X 0,Y 211.952,Z 522.185,A -85,B 0,C 180,E1 -20793.802,E2 -20793.802} C_VEL
LIN {X 0,Y 212.5,Z 520.398,A -85,B 0,C 180,E1 -20797.601,E2 -20797.601} C_VEL
LIN {X 0,Y 213.609,Z 517.345,A -85,B 0,C 180,E1 -20801.385,E2 -20801.385} C_VEL
LIN {X 0,Y 215.387,Z 512.939,A -85,B 0,C 180,E1 -20805.131,E2 -20805.131} C_VEL
LIN {X 0,Y 217.9,Z 507.029,A -85,B 0,C 180,E1 -20808.815,E2 -20808.815} C_VEL
LIN {X 0,Y 220.826,Z 500.467,A -85,B 0,C 180,E1 -20811.959,E2 -20811.959} C_VEL
LIN {X 0,Y 224.033,Z 492.391,A -85,B 0,C 180,E1 -20815.055,E2 -20815.055} C_VEL
LIN {X 0,Y 227.499,Z 484.02,A -85,B 0,C 180,E1 -20817.605,E2 -20817.605} C_VEL
LIN {X 0,Y 231.214,Z 473.982,A -85,B 0,C 180,E1 -20820.1,E2 -20820.1} C_VEL
LIN {X 0,Y 235.05,Z 462.853,A -85,B 0,C 180,E1 -20822.306,E2 -20822.306} C_VEL
LIN {X 0,Y 238.851,Z 450.389,A -85,B 0,C 180,E1 -20824.264,E2 -20824.264} C_VEL
LIN {X 0,Y 241.765,Z 438.398,A -85,B 0,C 180,E1 -20825.803,E2 -20825.803} C_VEL
LIN {X 0,Y 244.622,Z 425.056,A -85,B 0,C 180,E1 -20827.108,E2 -20827.108} C_VEL
LIN {X 0,Y 246.971,Z 411.283,A -85,B 0,C 180,E1 -20828.107,E2 -20828.107} C_VEL
LIN {X 0,Y 248.634,Z 397.175,A -85,B 0,C 180,E1 -20828.84,E2 -20828.84} C_VEL
LIN {X 0,Y 249.757,Z 381.191,A -85,B 0,C 180,E1 -20829.346,E2 -20829.346} C_VEL
LIN {X 0,Y 253.711,Z 303.16,A -85,B 0,C 180,E1 -20831.349,E2 -20831.349} C_VEL
LIN {X 0,Y 249.248,Z 292.728,A -85,B 0,C 180,E1 -20832.698,E2 -20832.698} C_VEL
LIN {X 0,Y 243.428,Z 280.917,A -85,B 0,C 180,E1 -20834.515,E2 -20834.515} C_VEL
LIN {X 0,Y 236.757,Z 268.91,A -85,B 0,C 180,E1 -20836.728,E2 -20836.728} C_VEL
LIN {X 0,Y 230.664,Z 259.079,A -85,B 0,C 180,E1 -20838.904,E2 -20838.904} C_VEL
LIN {X 0,Y 224.174,Z 249.39,A -85,B 0,C 180,E1 -20841.44,E2 -20841.44} C_VEL
LIN {X 0,Y 220.962,Z 244.472,A -85,B 0,C 180,E1 -20842.929,E2 -20842.929} C_VEL
LIN {X 0,Y 218.827,Z 238.378,A -85,B 0,C 180,E1 -20846.908,E2 -20846.908} C_VEL
LIN {X 0,Y 216.683,Z 232.935,A -85,B 0,C 180,E1 -20851.129,E2 -20851.129} C_VEL
LIN {X 0,Y 215.098,Z 228.749,A -85,B 0,C 180,E1 -20854.864,E2 -20854.864} C_VEL
LIN {X 0,Y 213.861,Z 225.527,A -85,B 0,C 180,E1 -20858.429,E2 -20858.429} C_VEL
LIN {X 0,Y 213.94,Z 225.453,A -85,B 0,C 180,E1 -20862.803,E2 -20862.803} C_VEL
LIN {X 0,Y 213.949,Z 225.454,A -85,B 0,C 180,E1 -20866.706,E2 -20866.706} C_VEL
LIN {X 0,Y 214.164,Z 225.432,A -85,B 0,C 180,E1 -20870.556,E2 -20870.556} C_VEL
LIN {X 0,Y 214.223,Z 225.41,A -85,B 0,C 180,E1 -20872.459,E2 -20872.459} C_VEL
LIN {X 0,Y 214.441,Z 225.39,A -85,B 0,C 180,E1 -20878.122,E2 -20878.122} C_VEL
LIN {X 0,Y 214.545,Z 225.375,A -85,B 0,C 180,E1 -20880,E2 -20880} C_VEL
LIN {X 0,Y 214.441,Z 225.384,A -85,B 0,C 180,E1 -20881.878,E2 -20881.878} C_VEL
LIN {X 0,Y 214.236,Z 225.425,A -85,B 0,C 180,E1 -20887.54,E2 -20887.54} C_VEL
LIN {X 0,Y 214.04,Z 225.444,A -85,B 0,C 180,E1 -20891.362,E2 -20891.362} C_VEL
LIN {X 0,Y 213.929,Z 225.455,A -85,B 0,C 180,E1 -20895.237,E2 -20895.237} C_VEL
LIN {X 0,Y 213.864,Z 225.572,A -85,B 0,C 180,E1 -20899.185,E2 -20899.185} C_VEL
LIN {X 0,Y 215.378,Z 229.246,A -85,B 0,C 180,E1 -20903.052,E2 -20903.052} C_VEL
LIN {X 0,Y 216.742,Z 232.582,A -85,B 0,C 180,E1 -20905.96,E2 -20905.96} C_VEL
LIN {X 0,Y 217.112,Z 233.877,A -85,B 0,C 180,E1 -20906.928,E2 -20906.928} C_VEL
LIN {X 0,Y 216.913,Z 235.769,A -85,B 0,C 180,E1 -20907.905,E2 -20907.905} C_VEL
LIN {X 0,Y 213.698,Z 243.497,A -85,B 0,C 180,E1 -20910.813,E2 -20910.813} C_VEL
LIN {X 0,Y 214.195,Z 245.055,A -85,B 0,C 180,E1 -20911.684,E2 -20911.684} C_VEL
LIN {X 0,Y 219.259,Z 252.215,A -85,B 0,C 180,E1 -20914.11,E2 -20914.11} C_VEL
LIN {X 0,Y 223.133,Z 257.83,A -85,B 0,C 180,E1 -20915.779,E2 -20915.779} C_VEL
LIN {X 0,Y 228.571,Z 266.096,A -85,B 0,C 180,E1 -20917.948,E2 -20917.948} C_VEL
LIN {X 0,Y 236.695,Z 280.185,A -85,B 0,C 180,E1 -20920.926,E2 -20920.926} C_VEL
LIN {X 0,Y 242.365,Z 291.074,A -85,B 0,C 180,E1 -20922.845,E2 -20922.845} C_VEL
LIN {X 0,Y 248.26,Z 304.078,A -85,B 0,C 180,E1 -20924.755,E2 -20924.755} C_VEL
LIN {X 0,Y 248.734,Z 305.209,A -85,B 0,C 180,E1 -20924.905,E2 -20924.905} C_VEL
LIN {X 0,Y 242.968,Z 401.693,A -85,B 0,C 180,E1 -20927.6,E2 -20927.6} C_VEL
LIN {X 0,Y 241.224,Z 416.785,A -85,B 0,C 180,E1 -20928.277,E2 -20928.277} C_VEL
LIN {X 0,Y 238.736,Z 431.401,A -85,B 0,C 180,E1 -20929.221,E2 -20929.221} C_VEL
LIN {X 0,Y 235.744,Z 445.132,A -85,B 0,C 180,E1 -20930.416,E2 -20930.416} C_VEL
LIN {X 0,Y 232.237,Z 458.725,A -85,B 0,C 180,E1 -20931.967,E2 -20931.967} C_VEL
LIN {X 0,Y 228.193,Z 472.085,A -85,B 0,C 180,E1 -20933.914,E2 -20933.914} C_VEL
LIN {X 0,Y 224.402,Z 483.341,A -85,B 0,C 180,E1 -20935.958,E2 -20935.958} C_VEL
LIN {X 0,Y 220.568,Z 493.763,A -85,B 0,C 180,E1 -20938.283,E2 -20938.283} C_VEL
LIN {X 0,Y 216.653,Z 504.106,A -85,B 0,C 180,E1 -20941.145,E2 -20941.145} C_VEL
LIN {X 0,Y 213.413,Z 512.766,A -85,B 0,C 180,E1 -20944.131,E2 -20944.131} C_VEL
LIN {X 0,Y 210.281,Z 520.512,A -85,B 0,C 180,E1 -20947.398,E2 -20947.398} C_VEL
LIN {X 0,Y 207.719,Z 527.462,A -85,B 0,C 180,E1 -20951.103,E2 -20951.103} C_VEL
LIN {X 0,Y 205.812,Z 533.312,A -85,B 0,C 180,E1 -20955.162,E2 -20955.162} C_VEL
LIN {X 0,Y 204.926,Z 536.558,A -85,B 0,C 180,E1 -20958.126,E2 -20958.126} C_VEL
LIN {X 0,Y 204.462,Z 539.75,A -85,B 0,C 180,E1 -20962.098,E2 -20962.098} C_VEL
LIN {X 0,Y 204.465,Z 541.433,A -85,B 0,C 180,E1 -20965.414,E2 -20965.414} C_VEL
LIN {X 0,Y 204.544,Z 542.14,A -85,B 0,C 180,E1 -20968.032,E2 -20968.032} C_VEL
LIN {X 0,Y 204.67,Z 542.305,A -85,B 0,C 180,E1 -20970.001,E2 -20970.001} C_VEL
LIN {X 0,Y 204.472,Z 541.643,A -85,B 0,C 180,E1 -20973.942,E2 -20973.942} C_VEL
LIN {X 0,Y 204.475,Z 540.839,A -85,B 0,C 180,E1 -20975.919,E2 -20975.919} C_VEL
LIN {X 0,Y 204.633,Z 538.275,A -85,B 0,C 180,E1 -20979.889,E2 -20979.889} C_VEL
LIN {X 0,Y 205.517,Z 534.411,A -85,B 0,C 180,E1 -20983.85,E2 -20983.85} C_VEL
LIN {X 0,Y 207.116,Z 529.149,A -85,B 0,C 180,E1 -20987.782,E2 -20987.782} C_VEL
LIN {X 0,Y 209.511,Z 522.352,A -85,B 0,C 180,E1 -20991.654,E2 -20991.654} C_VEL
LIN {X 0,Y 212.396,Z 514.98,A -85,B 0,C 180,E1 -20994.954,E2 -20994.954} C_VEL
LIN {X 0,Y 215.678,Z 506.581,A -85,B 0,C 180,E1 -20997.999,E2 -20997.999} C_VEL
LIN {X 0,Y 219.261,Z 496.926,A -85,B 0,C 180,E1 -21000.854,E2 -21000.854} C_VEL
LIN {X 0,Y 223.312,Z 486.092,A -85,B 0,C 180,E1 -21003.419,E2 -21003.419} C_VEL
LIN {X 0,Y 227.006,Z 475.382,A -85,B 0,C 180,E1 -21005.485,E2 -21005.485} C_VEL
LIN {X 0,Y 231.05,Z 462.539,A -85,B 0,C 180,E1 -21007.471,E2 -21007.471} C_VEL
LIN {X 0,Y 234.361,Z 450.044,A -85,B 0,C 180,E1 -21009.032,E2 -21009.032} C_VEL
LIN {X 0,Y 237.501,Z 436.527,A -85,B 0,C 180,E1 -21010.339,E2 -21010.339} C_VEL
LIN {X 0,Y 240.146,Z 422.934,A -85,B 0,C 180,E1 -21011.323,E2 -21011.323} C_VEL
LIN {X 0,Y 242.158,Z 408.591,A -85,B 0,C 180,E1 -21012.085,E2 -21012.085} C_VEL
LIN {X 0,Y 243.493,Z 392.666,A -85,B 0,C 180,E1 -21012.64,E2 -21012.64} C_VEL
LIN {X 0,Y 248.673,Z 305.218,A -85,B 0,C 180,E1 -21015.045,E2 -21015.045} C_VEL
LIN {X 0,Y 242.685,Z 291.896,A -85,B 0,C 180,E1 -21016.972,E2 -21016.972} C_VEL
LIN {X 0,Y 236.697,Z 280.175,A -85,B 0,C 180,E1 -21018.994,E2 -21018.994} C_VEL
LIN {X 0,Y 229.724,Z 268.218,A -85,B 0,C 180,E1 -21021.51,E2 -21021.51} C_VEL
LIN {X 0,Y 224.59,Z 260.074,A -85,B 0,C 180,E1 -21023.519,E2 -21023.519} C_VEL
LIN {X 0,Y 220.642,Z 254.175,A -85,B 0,C 180,E1 -21025.177,E2 -21025.177} C_VEL
LIN {X 0,Y 217.216,Z 249.398,A -85,B 0,C 180,E1 -21026.7,E2 -21026.7} C_VEL
LIN {X 0,Y 214.062,Z 244.782,A -85,B 0,C 180,E1 -21028.312,E2 -21028.312} C_VEL
LIN {X 0,Y 212.478,Z 240.384,A -85,B 0,C 180,E1 -21031.341,E2 -21031.341} C_VEL
LIN {X 0,Y 210.549,Z 235.693,A -85,B 0,C 180,E1 -21035.211,E2 -21035.211} C_VEL
LIN {X 0,Y 209.707,Z 233.323,A -85,B 0,C 180,E1 -21037.332,E2 -21037.332} C_VEL
LIN {X 0,Y 208.366,Z 229.989,A -85,B 0,C 180,E1 -21040.807,E2 -21040.807} C_VEL
LIN {X 0,Y 206.889,Z 226.412,A -85,B 0,C 180,E1 -21045.743,E2 -21045.743} C_VEL
LIN {X 0,Y 207.1,Z 226.298,A -85,B 0,C 180,E1 -21050.231,E2 -21050.231} C_VEL
LIN {X 0,Y 207.065,Z 226.302,A -85,B 0,C 180,E1 -21054.156,E2 -21054.156} C_VEL
LIN {X 0,Y 207.382,Z 226.264,A -85,B 0,C 180,E1 -21058.058,E2 -21058.058} C_VEL
LIN {X 0,Y 207.511,Z 226.25,A -85,B 0,C 180,E1 -21060,E2 -21060} C_VEL
LIN {X 0,Y 207.382,Z 226.268,A -85,B 0,C 180,E1 -21061.942,E2 -21061.942} C_VEL
LIN {X 0,Y 207.169,Z 226.289,A -85,B 0,C 180,E1 -21067.799,E2 -21067.799} C_VEL
LIN {X 0,Y 206.951,Z 226.316,A -85,B 0,C 180,E1 -21071.757,E2 -21071.757} C_VEL
LIN {X 0,Y 206.938,Z 226.515,A -85,B 0,C 180,E1 -21077.288,E2 -21077.288} C_VEL
LIN {X 0,Y 208.297,Z 229.886,A -85,B 0,C 180,E1 -21081.786,E2 -21081.786} C_VEL
LIN {X 0,Y 209.77,Z 233.713,A -85,B 0,C 180,E1 -21085.82,E2 -21085.82} C_VEL
LIN {X 0,Y 212.022,Z 239.516,A -85,B 0,C 180,E1 -21090.916,E2 -21090.916} C_VEL
LIN {X 0,Y 213.884,Z 244.703,A -85,B 0,C 180,E1 -21094.612,E2 -21094.612} C_VEL
LIN {X 0,Y 217.498,Z 249.833,A -85,B 0,C 180,E1 -21096.398,E2 -21096.398} C_VEL
LIN {X 0,Y 222.755,Z 257.599,A -85,B 0,C 180,E1 -21098.689,E2 -21098.689} C_VEL
LIN {X 0,Y 226.451,Z 263.222,A -85,B 0,C 180,E1 -21100.179,E2 -21100.179} C_VEL
LIN {X 0,Y 233.19,Z 274.237,A -85,B 0,C 180,E1 -21102.697,E2 -21102.697} C_VEL
LIN {X 0,Y 240.301,Z 287.627,A -85,B 0,C 180,E1 -21105.151,E2 -21105.151} C_VEL
LIN {X 0,Y 246.524,Z 300.842,A -85,B 0,C 180,E1 -21107.153,E2 -21107.153} C_VEL
LIN {X 0,Y 248.342,Z 305.107,A -85,B 0,C 180,E1 -21107.722,E2 -21107.722} C_VEL
LIN {X 0,Y 243.561,Z 392.372,A -85,B 0,C 180,E1 -21110.015,E2 -21110.015} C_VEL
LIN {X 0,Y 241.993,Z 407.136,A -85,B 0,C 180,E1 -21110.692,E2 -21110.692} C_VEL
LIN {X 0,Y 239.856,Z 420.909,A -85,B 0,C 180,E1 -21111.624,E2 -21111.624} C_VEL
LIN {X 0,Y 237.019,Z 434.33,A -85,B 0,C 180,E1 -21112.832,E2 -21112.832} C_VEL
LIN {X 0,Y 234.11,Z 446.156,A -85,B 0,C 180,E1 -21114.223,E2 -21114.223} C_VEL
LIN {X 0,Y 230.399,Z 459.097,A -85,B 0,C 180,E1 -21116.173,E2 -21116.173} C_VEL
LIN {X 0,Y 226.613,Z 469.96,A -85,B 0,C 180,E1 -21118.182,E2 -21118.182} C_VEL
LIN {X 0,Y 222.601,Z 480.73,A -85,B 0,C 180,E1 -21120.701,E2 -21120.701} C_VEL
LIN {X 0,Y 218.843,Z 489.697,A -85,B 0,C 180,E1 -21123.282,E2 -21123.282} C_VEL
LIN {X 0,Y 215.465,Z 497.723,A -85,B 0,C 180,E1 -21126.174,E2 -21126.174} C_VEL
LIN {X 0,Y 213.013,Z 503.478,A -85,B 0,C 180,E1 -21128.72,E2 -21128.72} C_VEL
LIN {X 0,Y 210.49,Z 508.73,A -85,B 0,C 180,E1 -21131.506,E2 -21131.506} C_VEL
LIN {X 0,Y 208.035,Z 514.304,A -85,B 0,C 180,E1 -21135.322,E2 -21135.322} C_VEL
LIN {X 0,Y 206.716,Z 517.547,A -85,B 0,C 180,E1 -21138.229,E2 -21138.229} C_VEL
LIN {X 0,Y 205.535,Z 520.642,A -85,B 0,C 180,E1 -21142.138,E2 -21142.138} C_VEL
LIN {X 0,Y 204.918,Z 522.475,A -85,B 0,C 180,E1 -21146.066,E2 -21146.066} C_VEL
LIN {X 0,Y 204.695,Z 523.096,A -85,B 0,C 180,E1 -21149.999,E2 -21149.999} C_VEL
LIN {X 0,Y 204.882,Z 522.517,A -85,B 0,C 180,E1 -21153.933,E2 -21153.933} C_VEL
LIN {X 0,Y 205.479,Z 520.73,A -85,B 0,C 180,E1 -21157.863,E2 -21157.863} C_VEL
LIN {X 0,Y 206.663,Z 517.677,A -85,B 0,C 180,E1 -21161.773,E2 -21161.773} C_VEL
LIN {X 0,Y 208.535,Z 513.273,A -85,B 0,C 180,E1 -21165.64,E2 -21165.64} C_VEL
LIN {X 0,Y 211.205,Z 507.367,A -85,B 0,C 180,E1 -21169.435,E2 -21169.435} C_VEL
LIN {X 0,Y 214.234,Z 500.809,A -85,B 0,C 180,E1 -21172.671,E2 -21172.671} C_VEL
LIN {X 0,Y 217.635,Z 492.74,A -85,B 0,C 180,E1 -21175.845,E2 -21175.845} C_VEL
LIN {X 0,Y 221.23,Z 484.373,A -85,B 0,C 180,E1 -21178.457,E2 -21178.457} C_VEL
LIN {X 0,Y 225.112,Z 474.348,A -85,B 0,C 180,E1 -21181.005,E2 -21181.005} C_VEL
LIN {X 0,Y 229.095,Z 463.24,A -85,B 0,C 180,E1 -21183.253,E2 -21183.253} C_VEL
LIN {X 0,Y 233.019,Z 450.808,A -85,B 0,C 180,E1 -21185.247,E2 -21185.247} C_VEL
LIN {X 0,Y 236.072,Z 438.858,A -85,B 0,C 180,E1 -21186.806,E2 -21186.806} C_VEL
LIN {X 0,Y 239.033,Z 425.583,A -85,B 0,C 180,E1 -21188.128,E2 -21188.128} C_VEL
LIN {X 0,Y 241.555,Z 411.162,A -85,B 0,C 180,E1 -21189.189,E2 -21189.189} C_VEL
LIN {X 0,Y 243.272,Z 396.899,A -85,B 0,C 180,E1 -21189.931,E2 -21189.931} C_VEL
LIN {X 0,Y 244.561,Z 378.795,A -85,B 0,C 180,E1 -21190.486,E2 -21190.486} C_VEL
LIN {X 0,Y 248.427,Z 305.205,A -85,B 0,C 180,E1 -21192.407,E2 -21192.407} C_VEL
LIN {X 0,Y 242.046,Z 290.945,A -85,B 0,C 180,E1 -21194.447,E2 -21194.447} C_VEL
LIN {X 0,Y 235.249,Z 277.889,A -85,B 0,C 180,E1 -21196.744,E2 -21196.744} C_VEL
LIN {X 0,Y 229.3,Z 267.781,A -85,B 0,C 180,E1 -21198.905,E2 -21198.905} C_VEL
LIN {X 0,Y 223.985,Z 259.477,A -85,B 0,C 180,E1 -21200.992,E2 -21200.992} C_VEL
LIN {X 0,Y 220.587,Z 254.376,A -85,B 0,C 180,E1 -21202.424,E2 -21202.424} C_VEL
LIN {X 0,Y 217.015,Z 249.273,A -85,B 0,C 180,E1 -21204.022,E2 -21204.022} C_VEL
LIN {X 0,Y 213.778,Z 244.476,A -85,B 0,C 180,E1 -21205.713,E2 -21205.713} C_VEL
LIN {X 0,Y 211.787,Z 239.185,A -85,B 0,C 180,E1 -21209.629,E2 -21209.629} C_VEL
LIN {X 0,Y 209.586,Z 233.275,A -85,B 0,C 180,E1 -21214.872,E2 -21214.872} C_VEL
LIN {X 0,Y 208.385,Z 230.157,A -85,B 0,C 180,E1 -21218.223,E2 -21218.223} C_VEL
LIN {X 0,Y 206.886,Z 226.398,A -85,B 0,C 180,E1 -21223.471,E2 -21223.471} C_VEL
LIN {X 0,Y 206.939,Z 226.318,A -85,B 0,C 180,E1 -21228.242,E2 -21228.242} C_VEL
LIN {X 0,Y 207.164,Z 226.29,A -85,B 0,C 180,E1 -21232.201,E2 -21232.201} C_VEL
LIN {X 0,Y 207.378,Z 226.268,A -85,B 0,C 180,E1 -21238.058,E2 -21238.058} C_VEL
LIN {X 0,Y 207.51,Z 226.251,A -85,B 0,C 180,E1 -21240,E2 -21240} C_VEL
LIN {X 0,Y 207.378,Z 226.264,A -85,B 0,C 180,E1 -21241.942,E2 -21241.942} C_VEL
LIN {X 0,Y 207.173,Z 226.304,A -85,B 0,C 180,E1 -21247.798,E2 -21247.798} C_VEL
LIN {X 0,Y 206.977,Z 226.328,A -85,B 0,C 180,E1 -21251.755,E2 -21251.755} C_VEL
LIN {X 0,Y 206.91,Z 226.492,A -85,B 0,C 180,E1 -21254.256,E2 -21254.256} C_VEL
LIN {X 0,Y 208.517,Z 230.675,A -85,B 0,C 180,E1 -21259.697,E2 -21259.697} C_VEL
LIN {X 0,Y 209.754,Z 233.467,A -85,B 0,C 180,E1 -21262.663,E2 -21262.663} C_VEL
LIN {X 0,Y 211.532,Z 238.121,A -85,B 0,C 180,E1 -21266.726,E2 -21266.726} C_VEL
LIN {X 0,Y 213.511,Z 243.231,A -85,B 0,C 180,E1 -21270.59,E2 -21270.59} C_VEL
LIN {X 0,Y 214.195,Z 245.055,A -85,B 0,C 180,E1 -21271.684,E2 -21271.684} C_VEL
LIN {X 0,Y 216.285,Z 248.677,A -85,B 0,C 180,E1 -21272.785,E2 -21272.785} C_VEL
LIN {X 0,Y 217.99,Z 253.198,A -85,B 0,C 180,E1 -21273.696,E2 -21273.696} C_VEL
LIN {X 0,Y 220.981,Z 263.1,A -85,B 0,C 180,E1 -21275.308,E2 -21275.308} C_VEL
LIN {X 0,Y 222.82,Z 267.684,A -85,B 0,C 180,E1 -21276.193,E2 -21276.193} C_VEL
LIN {X 0,Y 223.575,Z 269.047,A -85,B 0,C 180,E1 -21276.516,E2 -21276.516} C_VEL
LIN {X 0,Y 230.276,Z 280.384,A -85,B 0,C 180,E1 -21279.152,E2 -21279.152} C_VEL
LIN {X 0,Y 236.833,Z 292.837,A -85,B 0,C 180,E1 -21281.533,E2 -21281.533} C_VEL
LIN {X 0,Y 242.273,Z 304.702,A -85,B 0,C 180,E1 -21283.404,E2 -21283.404} C_VEL
LIN {X 0,Y 243.554,Z 307.674,A -85,B 0,C 180,E1 -21283.832,E2 -21283.832} C_VEL
LIN {X 0,Y 237.642,Z 402.008,A -85,B 0,C 180,E1 -21286.489,E2 -21286.489} C_VEL
LIN {X 0,Y 235.713,Z 417.672,A -85,B 0,C 180,E1 -21287.217,E2 -21287.217} C_VEL
LIN {X 0,Y 233.155,Z 432.004,A -85,B 0,C 180,E1 -21288.172,E2 -21288.172} C_VEL
LIN {X 0,Y 230.293,Z 444.652,A -85,B 0,C 180,E1 -21289.285,E2 -21289.285} C_VEL
LIN {X 0,Y 226.79,Z 457.742,A -85,B 0,C 180,E1 -21290.78,E2 -21290.78} C_VEL
LIN {X 0,Y 222.91,Z 470.465,A -85,B 0,C 180,E1 -21292.634,E2 -21292.634} C_VEL
LIN {X 0,Y 218.494,Z 482.963,A -85,B 0,C 180,E1 -21294.905,E2 -21294.905} C_VEL
LIN {X 0,Y 214.508,Z 493.394,A -85,B 0,C 180,E1 -21297.277,E2 -21297.277} C_VEL
LIN {X 0,Y 210.132,Z 504.399,A -85,B 0,C 180,E1 -21300.41,E2 -21300.41} C_VEL
LIN {X 0,Y 206.469,Z 513.624,A -85,B 0,C 180,E1 -21303.737,E2 -21303.737} C_VEL
LIN {X 0,Y 203.653,Z 520.166,A -85,B 0,C 180,E1 -21306.619,E2 -21306.619} C_VEL
LIN {X 0,Y 200.803,Z 527.516,A -85,B 0,C 180,E1 -21310.679,E2 -21310.679} C_VEL
LIN {X 0,Y 198.886,Z 532.973,A -85,B 0,C 180,E1 -21314.633,E2 -21314.633} C_VEL
LIN {X 0,Y 197.914,Z 536.221,A -85,B 0,C 180,E1 -21317.699,E2 -21317.699} C_VEL
LIN {X 0,Y 197.394,Z 539.416,A -85,B 0,C 180,E1 -21321.813,E2 -21321.813} C_VEL
LIN {X 0,Y 197.392,Z 541.325,A -85,B 0,C 180,E1 -21325.917,E2 -21325.917} C_VEL
LIN {X 0,Y 197.581,Z 541.972,A -85,B 0,C 180,E1 -21330.001,E2 -21330.001} C_VEL
LIN {X 0,Y 197.393,Z 541.31,A -85,B 0,C 180,E1 -21334.084,E2 -21334.084} C_VEL
LIN {X 0,Y 197.401,Z 539.38,A -85,B 0,C 180,E1 -21338.188,E2 -21338.188} C_VEL
LIN {X 0,Y 197.927,Z 536.17,A -85,B 0,C 180,E1 -21342.302,E2 -21342.302} C_VEL
LIN {X 0,Y 199.313,Z 531.622,A -85,B 0,C 180,E1 -21346.385,E2 -21346.385} C_VEL
LIN {X 0,Y 201.459,Z 525.609,A -85,B 0,C 180,E1 -21350.418,E2 -21350.418} C_VEL
LIN {X 0,Y 204.445,Z 517.975,A -85,B 0,C 180,E1 -21354.363,E2 -21354.363} C_VEL
LIN {X 0,Y 207.918,Z 509.75,A -85,B 0,C 180,E1 -21357.696,E2 -21357.696} C_VEL
LIN {X 0,Y 211.851,Z 499.806,A -85,B 0,C 180,E1 -21360.944,E2 -21360.944} C_VEL
LIN {X 0,Y 215.871,Z 489.566,A -85,B 0,C 180,E1 -21363.605,E2 -21363.605} C_VEL
LIN {X 0,Y 220.407,Z 477.321,A -85,B 0,C 180,E1 -21366.15,E2 -21366.15} C_VEL
LIN {X 0,Y 224.559,Z 464.952,A -85,B 0,C 180,E1 -21368.179,E2 -21368.179} C_VEL
LIN {X 0,Y 228.482,Z 451.056,A -85,B 0,C 180,E1 -21369.996,E2 -21369.996} C_VEL
LIN {X 0,Y 231.888,Z 437.112,A -85,B 0,C 180,E1 -21371.383,E2 -21371.383} C_VEL
LIN {X 0,Y 234.579,Z 423.763,A -85,B 0,C 180,E1 -21372.384,E2 -21372.384} C_VEL
LIN {X 0,Y 236.795,Z 408.819,A -85,B 0,C 180,E1 -21373.196,E2 -21373.196} C_VEL
LIN {X 0,Y 238.19,Z 393.112,A -85,B 0,C 180,E1 -21373.753,E2 -21373.753} C_VEL
LIN {X 0,Y 243.316,Z 307.268,A -85,B 0,C 180,E1 -21376.173,E2 -21376.173} C_VEL
LIN {X 0,Y 237.287,Z 293.831,A -85,B 0,C 180,E1 -21378.23,E2 -21378.23} C_VEL
LIN {X 0,Y 230.605,Z 281.081,A -85,B 0,C 180,E1 -21380.633,E2 -21380.633} C_VEL
LIN {X 0,Y 224.107,Z 269.969,A -85,B 0,C 180,E1 -21383.164,E2 -21383.164} C_VEL
LIN {X 0,Y 218.18,Z 260.694,A -85,B 0,C 180,E1 -21385.699,E2 -21385.699} C_VEL
LIN {X 0,Y 214.153,Z 254.959,A -85,B 0,C 180,E1 -21387.564,E2 -21387.564} C_VEL
LIN {X 0,Y 209.982,Z 249.236,A -85,B 0,C 180,E1 -21389.663,E2 -21389.663} C_VEL
LIN {X 0,Y 206.916,Z 244.785,A -85,B 0,C 180,E1 -21391.469,E2 -21391.469} C_VEL
LIN {X 0,Y 204.857,Z 239.722,A -85,B 0,C 180,E1 -21395.69,E2 -21395.69} C_VEL
LIN {X 0,Y 203.25,Z 235.652,A -85,B 0,C 180,E1 -21399.771,E2 -21399.771} C_VEL
LIN {X 0,Y 201.873,Z 232.37,A -85,B 0,C 180,E1 -21403.829,E2 -21403.829} C_VEL
LIN {X 0,Y 201.404,Z 230.908,A -85,B 0,C 180,E1 -21405.862,E2 -21405.862} C_VEL
LIN {X 0,Y 200.186,Z 227.79,A -85,B 0,C 180,E1 -21411.928,E2 -21411.928} C_VEL
LIN {X 0,Y 200.029,Z 227.243,A -85,B 0,C 180,E1 -21413.95,E2 -21413.95} C_VEL
LIN {X 0,Y 200.321,Z 227.144,A -85,B 0,C 180,E1 -21417.99,E2 -21417.99} C_VEL
LIN {X 0,Y 200.476,Z 227.126,A -85,B 0,C 180,E1 -21420,E2 -21420} C_VEL
LIN {X 0,Y 200.03,Z 227.179,A -85,B 0,C 180,E1 -21424.03,E2 -21424.03} C_VEL
LIN {X 0,Y 200.078,Z 227.267,A -85,B 0,C 180,E1 -21429.095,E2 -21429.095} C_VEL
LIN {X 0,Y 201.166,Z 230.566,A -85,B 0,C 180,E1 -21436.23,E2 -21436.23} C_VEL
LIN {X 0,Y 203.003,Z 235.052,A -85,B 0,C 180,E1 -21442.385,E2 -21442.385} C_VEL
LIN {X 0,Y 204.509,Z 239.182,A -85,B 0,C 180,E1 -21446.684,E2 -21446.684} C_VEL
LIN {X 0,Y 206.614,Z 244.605,A -85,B 0,C 180,E1 -21451.347,E2 -21451.347} C_VEL
LIN {X 0,Y 211.839,Z 251.825,A -85,B 0,C 180,E1 -21454.261,E2 -21454.261} C_VEL
LIN {X 0,Y 215.793,Z 257.456,A -85,B 0,C 180,E1 -21456.176,E2 -21456.176} C_VEL
LIN {X 0,Y 219.935,Z 263.704,A -85,B 0,C 180,E1 -21458.034,E2 -21458.034} C_VEL
LIN {X 0,Y 224.785,Z 271.236,A -85,B 0,C 180,E1 -21460.041,E2 -21460.041} C_VEL
LIN {X 0,Y 231.897,Z 283.735,A -85,B 0,C 180,E1 -21462.759,E2 -21462.759} C_VEL
LIN {X 0,Y 238.849,Z 297.679,A -85,B 0,C 180,E1 -21465.201,E2 -21465.201} C_VEL
LIN {X 0,Y 243.16,Z 307.533,A -85,B 0,C 180,E1 -21466.64,E2 -21466.64} C_VEL
LIN {X 0,Y 238.293,Z 392.335,A -85,B 0,C 180,E1 -21468.888,E2 -21468.888} C_VEL
LIN {X 0,Y 236.682,Z 407.036,A -85,B 0,C 180,E1 -21469.562,E2 -21469.562} C_VEL
LIN {X 0,Y 234.588,Z 420.315,A -85,B 0,C 180,E1 -21470.459,E2 -21470.459} C_VEL
LIN {X 0,Y 231.889,Z 432.999,A -85,B 0,C 180,E1 -21471.588,E2 -21471.588} C_VEL
LIN {X 0,Y 228.622,Z 445.705,A -85,B 0,C 180,E1 -21473.06,E2 -21473.06} C_VEL
LIN {X 0,Y 224.93,Z 458.333,A -85,B 0,C 180,E1 -21474.961,E2 -21474.961} C_VEL
LIN {X 0,Y 220.608,Z 470.337,A -85,B 0,C 180,E1 -21477.209,E2 -21477.209} C_VEL
LIN {X 0,Y 216.444,Z 481.092,A -85,B 0,C 180,E1 -21479.782,E2 -21479.782} C_VEL
LIN {X 0,Y 212.538,Z 490.048,A -85,B 0,C 180,E1 -21482.423,E2 -21482.423} C_VEL
LIN {X 0,Y 208.814,Z 498.43,A -85,B 0,C 180,E1 -21485.541,E2 -21485.541} C_VEL
LIN {X 0,Y 206.428,Z 503.819,A -85,B 0,C 180,E1 -21488.006,E2 -21488.006} C_VEL
LIN {X 0,Y 203.019,Z 510.642,A -85,B 0,C 180,E1 -21491.846,E2 -21491.846} C_VEL
LIN {X 0,Y 200.673,Z 515.833,A -85,B 0,C 180,E1 -21495.808,E2 -21495.808} C_VEL
LIN {X 0,Y 199.039,Z 519.592,A -85,B 0,C 180,E1 -21499.831,E2 -21499.831} C_VEL
LIN {X 0,Y 198.088,Z 522.047,A -85,B 0,C 180,E1 -21503.889,E2 -21503.889} C_VEL
LIN {X 0,Y 197.661,Z 523.269,A -85,B 0,C 180,E1 -21507.962,E2 -21507.962} C_VEL
LIN {X 0,Y 197.652,Z 523.289,A -85,B 0,C 180,E1 -21512.037,E2 -21512.037} C_VEL
LIN {X 0,Y 198.039,Z 522.111,A -85,B 0,C 180,E1 -21516.111,E2 -21516.111} C_VEL
LIN {X 0,Y 198.98,Z 519.7,A -85,B 0,C 180,E1 -21520.171,E2 -21520.171} C_VEL
LIN {X 0,Y 200.609,Z 515.984,A -85,B 0,C 180,E1 -21524.195,E2 -21524.195} C_VEL
LIN {X 0,Y 202.946,Z 510.86,A -85,B 0,C 180,E1 -21528.159,E2 -21528.159} C_VEL
LIN {X 0,Y 206.329,Z 504.112,A -85,B 0,C 180,E1 -21532.004,E2 -21532.004} C_VEL
LIN {X 0,Y 209.59,Z 496.755,A -85,B 0,C 180,E1 -21535.3,E2 -21535.3} C_VEL
LIN {X 0,Y 213.049,Z 489.096,A -85,B 0,C 180,E1 -21538.038,E2 -21538.038} C_VEL
LIN {X 0,Y 217.011,Z 479.949,A -85,B 0,C 180,E1 -21540.667,E2 -21540.667} C_VEL
LIN {X 0,Y 220.486,Z 470.884,A -85,B 0,C 180,E1 -21542.81,E2 -21542.81} C_VEL
LIN {X 0,Y 224.82,Z 458.985,A -85,B 0,C 180,E1 -21545.057,E2 -21545.057} C_VEL
LIN {X 0,Y 228.71,Z 445.963,A -85,B 0,C 180,E1 -21547.031,E2 -21547.031} C_VEL
LIN {X 0,Y 231.807,Z 434.038,A -85,B 0,C 180,E1 -21548.426,E2 -21548.426} C_VEL
LIN {X 0,Y 234.671,Z 420.457,A -85,B 0,C 180,E1 -21549.662,E2 -21549.662} C_VEL
LIN {X 0,Y 237.025,Z 405.516,A -85,B 0,C 180,E1 -21550.645,E2 -21550.645} C_VEL
LIN {X 0,Y 238.482,Z 391.837,A -85,B 0,C 180,E1 -21551.251,E2 -21551.251} C_VEL
LIN {X 0,Y 243.212,Z 307.496,A -85,B 0,C 180,E1 -21553.506,E2 -21553.506} C_VEL
LIN {X 0,Y 237.361,Z 294.306,A -85,B 0,C 180,E1 -21555.482,E2 -21555.482} C_VEL
LIN {X 0,Y 229.834,Z 279.807,A -85,B 0,C 180,E1 -21558.186,E2 -21558.186} C_VEL
LIN {X 0,Y 223.239,Z 268.841,A -85,B 0,C 180,E1 -21560.766,E2 -21560.766} C_VEL
LIN {X 0,Y 217.772,Z 260.304,A -85,B 0,C 180,E1 -21563.125,E2 -21563.125} C_VEL
LIN {X 0,Y 214.021,Z 254.902,A -85,B 0,C 180,E1 -21564.874,E2 -21564.874} C_VEL
LIN {X 0,Y 210.195,Z 249.593,A -85,B 0,C 180,E1 -21566.802,E2 -21566.802} C_VEL
LIN {X 0,Y 206.582,Z 244.576,A -85,B 0,C 180,E1 -21568.913,E2 -21568.913} C_VEL
LIN {X 0,Y 204.527,Z 239.317,A -85,B 0,C 180,E1 -21573.467,E2 -21573.467} C_VEL
LIN {X 0,Y 203.793,Z 237.194,A -85,B 0,C 180,E1 -21575.554,E2 -21575.554} C_VEL
LIN {X 0,Y 202.348,Z 233.703,A -85,B 0,C 180,E1 -21579.676,E2 -21579.676} C_VEL
LIN {X 0,Y 201.316,Z 230.771,A -85,B 0,C 180,E1 -21583.782,E2 -21583.782} C_VEL
LIN {X 0,Y 200.1,Z 227.369,A -85,B 0,C 180,E1 -21591.161,E2 -21591.161} C_VEL
LIN {X 0,Y 200.027,Z 227.18,A -85,B 0,C 180,E1 -21595.97,E2 -21595.97} C_VEL
LIN {X 0,Y 200.475,Z 227.127,A -85,B 0,C 180,E1 -21600,E2 -21600} C_VEL
LIN {X 0,Y 200.031,Z 227.212,A -85,B 0,C 180,E1 -21604.029,E2 -21604.029} C_VEL
LIN {X 0,Y 200.158,Z 227.626,A -85,B 0,C 180,E1 -21607.059,E2 -21607.059} C_VEL
LIN {X 0,Y 200.878,Z 230.024,A -85,B 0,C 180,E1 -21612.117,E2 -21612.117} C_VEL
LIN {X 0,Y 201.512,Z 231.082,A -85,B 0,C 180,E1 -21614.13,E2 -21614.13} C_VEL
LIN {X 0,Y 202.633,Z 234.058,A -85,B 0,C 180,E1 -21618.189,E2 -21618.189} C_VEL
LIN {X 0,Y 204.51,Z 238.772,A -85,B 0,C 180,E1 -21623.278,E2 -21623.278} C_VEL
LIN {X 0,Y 205.848,Z 242.194,A -85,B 0,C 180,E1 -21626.349,E2 -21626.349} C_VEL
LIN {X 0,Y 207.111,Z 245.186,A -85,B 0,C 180,E1 -21628.571,E2 -21628.571} C_VEL
LIN {X 0,Y 212.444,Z 252.531,A -85,B 0,C 180,E1 -21631.47,E2 -21631.47} C_VEL
LIN {X 0,Y 216.281,Z 257.938,A -85,B 0,C 180,E1 -21633.323,E2 -21633.323} C_VEL
LIN {X 0,Y 220.04,Z 263.535,A -85,B 0,C 180,E1 -21635.018,E2 -21635.018} C_VEL
LIN {X 0,Y 223.575,Z 269.047,A -85,B 0,C 180,E1 -21636.516,E2 -21636.516} C_VEL
LIN {X 0,Y 224.771,Z 272.196,A -85,B 0,C 180,E1 -21637.066,E2 -21637.066} C_VEL
LIN {X 0,Y 226.542,Z 284.824,A -85,B 0,C 180,E1 -21638.258,E2 -21638.258} C_VEL
LIN {X 0,Y 227.869,Z 287.854,A -85,B 0,C 180,E1 -21638.808,E2 -21638.808} C_VEL
LIN {X 0,Y 233.772,Z 299.466,A -85,B 0,C 180,E1 -21641.025,E2 -21641.025} C_VEL
LIN {X 0,Y 238.332,Z 309.832,A -85,B 0,C 180,E1 -21642.666,E2 -21642.666} C_VEL
LIN {X 0,Y 236.075,Z 346.031,A -85,B 0,C 180,E1 -21643.692,E2 -21643.692} C_VEL
LIN {X 0,Y 232.406,Z 402.274,A -85,B 0,C 180,E1 -21645.327,E2 -21645.327} C_VEL
LIN {X 0,Y 230.531,Z 417.028,A -85,B 0,C 180,E1 -21646.013,E2 -21646.013} C_VEL
LIN {X 0,Y 227.863,Z 431.47,A -85,B 0,C 180,E1 -21646.97,E2 -21646.97} C_VEL
LIN {X 0,Y 224.456,Z 445.987,A -85,B 0,C 180,E1 -21648.291,E2 -21648.291} C_VEL
LIN {X 0,Y 221.012,Z 458.321,A -85,B 0,C 180,E1 -21649.745,E2 -21649.745} C_VEL
LIN {X 0,Y 216.846,Z 471.3,A -85,B 0,C 180,E1 -21651.697,E2 -21651.697} C_VEL
LIN {X 0,Y 212.273,Z 483.582,A -85,B 0,C 180,E1 -21654.009,E2 -21654.009} C_VEL
LIN {X 0,Y 207.795,Z 494.734,A -85,B 0,C 180,E1 -21656.662,E2 -21656.662} C_VEL
LIN {X 0,Y 203.582,Z 504.773,A -85,B 0,C 180,E1 -21659.66,E2 -21659.66} C_VEL
LIN {X 0,Y 200.028,Z 513.276,A -85,B 0,C 180,E1 -21662.823,E2 -21662.823} C_VEL
LIN {X 0,Y 197.058,Z 519.821,A -85,B 0,C 180,E1 -21665.787,E2 -21665.787} C_VEL
LIN {X 0,Y 194.026,Z 527.188,A -85,B 0,C 180,E1 -21669.984,E2 -21669.984} C_VEL
LIN {X 0,Y 191.969,Z 532.634,A -85,B 0,C 180,E1 -21674.064,E2 -21674.064} C_VEL
LIN {X 0,Y 190.912,Z 535.884,A -85,B 0,C 180,E1 -21677.24,E2 -21677.24} C_VEL
LIN {X 0,Y 190.32,Z 539.08,A -85,B 0,C 180,E1 -21681.507,E2 -21681.507} C_VEL
LIN {X 0,Y 190.314,Z 540.993,A -85,B 0,C 180,E1 -21685.765,E2 -21685.765} C_VEL
LIN {X 0,Y 190.495,Z 541.64,A -85,B 0,C 180,E1 -21690.001,E2 -21690.001} C_VEL
LIN {X 0,Y 190.329,Z 540.921,A -85,B 0,C 180,E1 -21694.451,E2 -21694.451} C_VEL
LIN {X 0,Y 190.326,Z 539.044,A -85,B 0,C 180,E1 -21698.495,E2 -21698.495} C_VEL
LIN {X 0,Y 190.927,Z 535.832,A -85,B 0,C 180,E1 -21702.76,E2 -21702.76} C_VEL
LIN {X 0,Y 192.441,Z 531.282,A -85,B 0,C 180,E1 -21706.988,E2 -21706.988} C_VEL
LIN {X 0,Y 194.733,Z 525.265,A -85,B 0,C 180,E1 -21711.156,E2 -21711.156} C_VEL
LIN {X 0,Y 197.925,Z 517.628,A -85,B 0,C 180,E1 -21715.221,E2 -21715.221} C_VEL
LIN {X 0,Y 201.563,Z 509.396,A -85,B 0,C 180,E1 -21718.648,E2 -21718.648} C_VEL
LIN {X 0,Y 205.717,Z 499.444,A -85,B 0,C 180,E1 -21721.974,E2 -21721.974} C_VEL
LIN {X 0,Y 209.956,Z 489.193,A -85,B 0,C 180,E1 -21724.685,E2 -21724.685} C_VEL
LIN {X 0,Y 214.262,Z 478.013,A -85,B 0,C 180,E1 -21727.065,E2 -21727.065} C_VEL
LIN {X 0,Y 218.551,Z 465.842,A -85,B 0,C 180,E1 -21729.131,E2 -21729.131} C_VEL
LIN {X 0,Y 222.5,Z 452.603,A -85,B 0,C 180,E1 -21730.934,E2 -21730.934} C_VEL
LIN {X 0,Y 226.085,Z 438.692,A -85,B 0,C 180,E1 -21732.39,E2 -21732.39} C_VEL
LIN {X 0,Y 229.091,Z 424.48,A -85,B 0,C 180,E1 -21733.498,E2 -21733.498} C_VEL
LIN {X 0,Y 231.407,Z 409.947,A -85,B 0,C 180,E1 -21734.309,E2 -21734.309} C_VEL
LIN {X 0,Y 232.851,Z 395.153,A -85,B 0,C 180,E1 -21734.871,E2 -21734.871} C_VEL
LIN {X 0,Y 238.26,Z 309.813,A -85,B 0,C 180,E1 -21737.279,E2 -21737.279} C_VEL
LIN {X 0,Y 231.932,Z 295.784,A -85,B 0,C 180,E1 -21739.566,E2 -21739.566} C_VEL
LIN {X 0,Y 226.059,Z 284.562,A -85,B 0,C 180,E1 -21741.812,E2 -21741.812} C_VEL
LIN {X 0,Y 220.305,Z 274.624,A -85,B 0,C 180,E1 -21744.184,E2 -21744.184} C_VEL
LIN {X 0,Y 214.757,Z 265.768,A -85,B 0,C 180,E1 -21746.69,E2 -21746.69} C_VEL
LIN {X 0,Y 211.256,Z 260.687,A -85,B 0,C 180,E1 -21748.394,E2 -21748.394} C_VEL
LIN {X 0,Y 207.395,Z 255.233,A -85,B 0,C 180,E1 -21750.431,E2 -21750.431} C_VEL
LIN {X 0,Y 203.735,Z 250.247,A -85,B 0,C 180,E1 -21752.545,E2 -21752.545} C_VEL
LIN {X 0,Y 200.205,Z 245.674,A -85,B 0,C 180,E1 -21754.809,E2 -21754.809} C_VEL
LIN {X 0,Y 199.492,Z 244.465,A -85,B 0,C 180,E1 -21755.548,E2 -21755.548} C_VEL
LIN {X 0,Y 198.034,Z 240.807,A -85,B 0,C 180,E1 -21759.214,E2 -21759.214} C_VEL
LIN {X 0,Y 196.656,Z 237.403,A -85,B 0,C 180,E1 -21763.388,E2 -21763.388} C_VEL
LIN {X 0,Y 196.158,Z 235.919,A -85,B 0,C 180,E1 -21765.476,E2 -21765.476} C_VEL
LIN {X 0,Y 194.923,Z 232.668,A -85,B 0,C 180,E1 -21771.708,E2 -21771.708} C_VEL
LIN {X 0,Y 194.672,Z 231.905,A -85,B 0,C 180,E1 -21773.783,E2 -21773.783} C_VEL
LIN {X 0,Y 194.35,Z 230.697,A -85,B 0,C 180,E1 -21780,E2 -21780} C_VEL
LIN {X 0,Y 194.299,Z 231.346,A -85,B 0,C 180,E1 -21786.23,E2 -21786.23} C_VEL
LIN {X 0,Y 194.61,Z 231.725,A -85,B 0,C 180,E1 -21788.306,E2 -21788.306} C_VEL
LIN {X 0,Y 194.934,Z 233.43,A -85,B 0,C 180,E1 -21792.493,E2 -21792.493} C_VEL
LIN {X 0,Y 195.902,Z 235.528,A -85,B 0,C 180,E1 -21796.679,E2 -21796.679} C_VEL
LIN {X 0,Y 197.728,Z 240.197,A -85,B 0,C 180,E1 -21803.016,E2 -21803.016} C_VEL
LIN {X 0,Y 199.371,Z 244.595,A -85,B 0,C 180,E1 -21807.481,E2 -21807.481} C_VEL
LIN {X 0,Y 203.134,Z 249.626,A -85,B 0,C 180,E1 -21810.068,E2 -21810.068} C_VEL
LIN {X 0,Y 209.029,Z 257.57,A -85,B 0,C 180,E1 -21813.406,E2 -21813.406} C_VEL
LIN {X 0,Y 212.864,Z 263.177,A -85,B 0,C 180,E1 -21815.355,E2 -21815.355} C_VEL
LIN {X 0,Y 216.91,Z 269.423,A -85,B 0,C 180,E1 -21817.256,E2 -21817.256} C_VEL
LIN {X 0,Y 221.38,Z 276.565,A -85,B 0,C 180,E1 -21819.195,E2 -21819.195} C_VEL
LIN {X 0,Y 228.073,Z 288.561,A -85,B 0,C 180,E1 -21821.878,E2 -21821.878} C_VEL
LIN {X 0,Y 234.364,Z 301.429,A -85,B 0,C 180,E1 -21824.205,E2 -21824.205} C_VEL
LIN {X 0,Y 238.026,Z 309.847,A -85,B 0,C 180,E1 -21825.496,E2 -21825.496} C_VEL
LIN {X 0,Y 233.017,Z 393.485,A -85,B 0,C 180,E1 -21827.758,E2 -21827.758} C_VEL
LIN {X 0,Y 231.362,Z 407.702,A -85,B 0,C 180,E1 -21828.43,E2 -21828.43} C_VEL
LIN {X 0,Y 228.936,Z 421.996,A -85,B 0,C 180,E1 -21829.426,E2 -21829.426} C_VEL
LIN {X 0,Y 225.923,Z 435.273,A -85,B 0,C 180,E1 -21830.667,E2 -21830.667} C_VEL
LIN {X 0,Y 222.544,Z 447.769,A -85,B 0,C 180,E1 -21832.2,E2 -21832.2} C_VEL
LIN {X 0,Y 218.787,Z 459.89,A -85,B 0,C 180,E1 -21834.109,E2 -21834.109} C_VEL
LIN {X 0,Y 214.67,Z 470.714,A -85,B 0,C 180,E1 -21836.182,E2 -21836.182} C_VEL
LIN {X 0,Y 210.332,Z 481.454,A -85,B 0,C 180,E1 -21838.807,E2 -21838.807} C_VEL
LIN {X 0,Y 206.269,Z 490.4,A -85,B 0,C 180,E1 -21841.509,E2 -21841.509} C_VEL
LIN {X 0,Y 202.6,Z 498.129,A -85,B 0,C 180,E1 -21844.412,E2 -21844.412} C_VEL
LIN {X 0,Y 199.877,Z 504.162,A -85,B 0,C 180,E1 -21847.245,E2 -21847.245} C_VEL
LIN {X 0,Y 196.272,Z 510.982,A -85,B 0,C 180,E1 -21851.199,E2 -21851.199} C_VEL
LIN {X 0,Y 193.789,Z 516.169,A -85,B 0,C 180,E1 -21855.293,E2 -21855.293} C_VEL
LIN {X 0,Y 192.066,Z 519.925,A -85,B 0,C 180,E1 -21859.457,E2 -21859.457} C_VEL
LIN {X 0,Y 191.053,Z 522.379,A -85,B 0,C 180,E1 -21863.663,E2 -21863.663} C_VEL
LIN {X 0,Y 190.583,Z 523.602,A -85,B 0,C 180,E1 -21867.886,E2 -21867.886} C_VEL
LIN {X 0,Y 190.573,Z 523.621,A -85,B 0,C 180,E1 -21872.113,E2 -21872.113} C_VEL
LIN {X 0,Y 190.993,Z 522.443,A -85,B 0,C 180,E1 -21876.337,E2 -21876.337} C_VEL
LIN {X 0,Y 191.983,Z 520.034,A -85,B 0,C 180,E1 -21880.546,E2 -21880.546} C_VEL
LIN {X 0,Y 193.719,Z 516.318,A -85,B 0,C 180,E1 -21884.711,E2 -21884.711} C_VEL
LIN {X 0,Y 196.198,Z 511.196,A -85,B 0,C 180,E1 -21888.806,E2 -21888.806} C_VEL
LIN {X 0,Y 199.768,Z 504.451,A -85,B 0,C 180,E1 -21892.766,E2 -21892.766} C_VEL
LIN {X 0,Y 203.08,Z 497.336,A -85,B 0,C 180,E1 -21896.063,E2 -21896.063} C_VEL
LIN {X 0,Y 206.807,Z 489.445,A -85,B 0,C 180,E1 -21898.963,E2 -21898.963} C_VEL
LIN {X 0,Y 210.95,Z 480.305,A -85,B 0,C 180,E1 -21901.649,E2 -21901.649} C_VEL
LIN {X 0,Y 215.427,Z 469.301,A -85,B 0,C 180,E1 -21904.245,E2 -21904.245} C_VEL
LIN {X 0,Y 219.485,Z 458.198,A -85,B 0,C 180,E1 -21906.325,E2 -21906.325} C_VEL
LIN {X 0,Y 223.282,Z 445.745,A -85,B 0,C 180,E1 -21908.21,E2 -21908.21} C_VEL
LIN {X 0,Y 226.752,Z 432.632,A -85,B 0,C 180,E1 -21909.735,E2 -21909.735} C_VEL
LIN {X 0,Y 229.503,Z 419.784,A -85,B 0,C 180,E1 -21910.885,E2 -21910.885} C_VEL
LIN {X 0,Y 231.833,Z 405.329,A -85,B 0,C 180,E1 -21911.829,E2 -21911.829} C_VEL
LIN {X 0,Y 233.32,Z 391.698,A -85,B 0,C 180,E1 -21912.432,E2 -21912.432} C_VEL
LIN {X 0,Y 238.13,Z 310.741,A -85,B 0,C 180,E1 -21914.604,E2 -21914.604} C_VEL
LIN {X 0,Y 237.824,Z 309.202,A -85,B 0,C 180,E1 -21914.744,E2 -21914.744} C_VEL
LIN {X 0,Y 232.903,Z 298.136,A -85,B 0,C 180,E1 -21916.497,E2 -21916.497} C_VEL
LIN {X 0,Y 226.724,Z 285.952,A -85,B 0,C 180,E1 -21918.827,E2 -21918.827} C_VEL
LIN {X 0,Y 220.755,Z 275.508,A -85,B 0,C 180,E1 -21921.26,E2 -21921.26} C_VEL
LIN {X 0,Y 214.817,Z 266.044,A -85,B 0,C 180,E1 -21923.921,E2 -21923.921} C_VEL
LIN {X 0,Y 211.14,Z 260.61,A -85,B 0,C 180,E1 -21925.718,E2 -21925.718} C_VEL
LIN {X 0,Y 207.438,Z 255.343,A -85,B 0,C 180,E1 -21927.679,E2 -21927.679} C_VEL
LIN {X 0,Y 203.4,Z 249.988,A -85,B 0,C 180,E1 -21930.016,E2 -21930.016} C_VEL
LIN {X 0,Y 199.285,Z 244.481,A -85,B 0,C 180,E1 -21932.884,E2 -21932.884} C_VEL
LIN {X 0,Y 198.591,Z 242.358,A -85,B 0,C 180,E1 -21934.87,E2 -21934.87} C_VEL
LIN {X 0,Y 197.111,Z 238.755,A -85,B 0,C 180,E1 -21939.111,E2 -21939.111} C_VEL
LIN {X 0,Y 196.018,Z 235.765,A -85,B 0,C 180,E1 -21943.331,E2 -21943.331} C_VEL
LIN {X 0,Y 194.881,Z 232.688,A -85,B 0,C 180,E1 -21949.611,E2 -21949.611} C_VEL
LIN {X 0,Y 194.743,Z 231.93,A -85,B 0,C 180,E1 -21951.7,E2 -21951.7} C_VEL
LIN {X 0,Y 194.335,Z 230.993,A -85,B 0,C 180,E1 -21957.927,E2 -21957.927} C_VEL
LIN {X 0,Y 194.479,Z 230.889,A -85,B 0,C 180,E1 -21960,E2 -21960} C_VEL
LIN {X 0,Y 194.774,Z 232.106,A -85,B 0,C 180,E1 -21966.214,E2 -21966.214} C_VEL
LIN {X 0,Y 195.275,Z 233.861,A -85,B 0,C 180,E1 -21970.367,E2 -21970.367} C_VEL
LIN {X 0,Y 196.315,Z 236.348,A -85,B 0,C 180,E1 -21974.858,E2 -21974.858} C_VEL
LIN {X 0,Y 197.401,Z 239.163,A -85,B 0,C 180,E1 -21978.688,E2 -21978.688} C_VEL
LIN {X 0,Y 199.515,Z 244.502,A -85,B 0,C 180,E1 -21984.31,E2 -21984.31} C_VEL
LIN {X 0,Y 200.896,Z 246.74,A -85,B 0,C 180,E1 -21985.514,E2 -21985.514} C_VEL
LIN {X 0,Y 205.158,Z 252.127,A -85,B 0,C 180,E1 -21988.149,E2 -21988.149} C_VEL
LIN {X 0,Y 209.811,Z 258.55,A -85,B 0,C 180,E1 -21990.728,E2 -21990.728} C_VEL
LIN {X 0,Y 214.183,Z 264.903,A -85,B 0,C 180,E1 -21992.92,E2 -21992.92} C_VEL
LIN {X 0,Y 219.358,Z 272.88,A -85,B 0,C 180,E1 -21995.289,E2 -21995.289} C_VEL
LIN {X 0,Y 225.386,Z 283.35,A -85,B 0,C 180,E1 -21997.828,E2 -21997.828} C_VEL
LIN {X 0,Y 227.869,Z 287.854,A -85,B 0,C 180,E1 -21998.808,E2 -21998.808} C_VEL
LIN {X 0,Y 228.991,Z 290.326,A -85,B 0,C 180,E1 -21999.259,E2 -21999.259} C_VEL
LIN {X 0,Y 229.682,Z 294.639,A -85,B 0,C 180,E1 -21999.666,E2 -21999.666} C_VEL
LIN {X 0,Y 230.251,Z 303.932,A -85,B 0,C 180,E1 -22000.269,E2 -22000.269} C_VEL
LIN {X 0,Y 231.231,Z 307.464,A -85,B 0,C 180,E1 -22000.706,E2 -22000.706} C_VEL
LIN {X 0,Y 233.338,Z 312.387,A -85,B 0,C 180,E1 -22001.5,E2 -22001.5} C_VEL
LIN {X 0,Y 227.409,Z 401.378,A -85,B 0,C 180,E1 -22004.068,E2 -22004.068} C_VEL
LIN {X 0,Y 225.423,Z 416.376,A -85,B 0,C 180,E1 -22004.747,E2 -22004.747} C_VEL
LIN {X 0,Y 222.717,Z 430.941,A -85,B 0,C 180,E1 -22005.721,E2 -22005.721} C_VEL
LIN {X 0,Y 219.186,Z 445.523,A -85,B 0,C 180,E1 -22007.052,E2 -22007.052} C_VEL
LIN {X 0,Y 215.262,Z 458.973,A -85,B 0,C 180,E1 -22008.669,E2 -22008.669} C_VEL
LIN {X 0,Y 210.816,Z 472.09,A -85,B 0,C 180,E1 -22010.7,E2 -22010.7} C_VEL
LIN {X 0,Y 206.527,Z 483.208,A -85,B 0,C 180,E1 -22012.843,E2 -22012.843} C_VEL
LIN {X 0,Y 201.845,Z 494.373,A -85,B 0,C 180,E1 -22015.543,E2 -22015.543} C_VEL
LIN {X 0,Y 197.484,Z 504.244,A -85,B 0,C 180,E1 -22018.543,E2 -22018.543} C_VEL
LIN {X 0,Y 193.659,Z 512.93,A -85,B 0,C 180,E1 -22021.852,E2 -22021.852} C_VEL
LIN {X 0,Y 190.515,Z 519.476,A -85,B 0,C 180,E1 -22024.899,E2 -22024.899} C_VEL
LIN {X 0,Y 187.349,Z 526.68,A -85,B 0,C 180,E1 -22029.124,E2 -22029.124} C_VEL
LIN {X 0,Y 185.063,Z 532.295,A -85,B 0,C 180,E1 -22033.453,E2 -22033.453} C_VEL
LIN {X 0,Y 183.923,Z 535.548,A -85,B 0,C 180,E1 -22036.747,E2 -22036.747} C_VEL
LIN {X 0,Y 183.241,Z 538.745,A -85,B 0,C 180,E1 -22041.176,E2 -22041.176} C_VEL
LIN {X 0,Y 183.226,Z 540.659,A -85,B 0,C 180,E1 -22045.601,E2 -22045.601} C_VEL
LIN {X 0,Y 183.41,Z 541.307,A -85,B 0,C 180,E1 -22050.001,E2 -22050.001} C_VEL
LIN {X 0,Y 183.231,Z 540.643,A -85,B 0,C 180,E1 -22054.4,E2 -22054.4} C_VEL
LIN {X 0,Y 183.247,Z 538.707,A -85,B 0,C 180,E1 -22058.825,E2 -22058.825} C_VEL
LIN {X 0,Y 183.939,Z 535.494,A -85,B 0,C 180,E1 -22063.254,E2 -22063.254} C_VEL
LIN {X 0,Y 185.59,Z 530.942,A -85,B 0,C 180,E1 -22067.635,E2 -22067.635} C_VEL
LIN {X 0,Y 188.028,Z 524.921,A -85,B 0,C 180,E1 -22071.949,E2 -22071.949} C_VEL
LIN {X 0,Y 191.46,Z 517.282,A -85,B 0,C 180,E1 -22076.136,E2 -22076.136} C_VEL
LIN {X 0,Y 195.291,Z 509.043,A -85,B 0,C 180,E1 -22079.659,E2 -22079.659} C_VEL
LIN {X 0,Y 198.993,Z 500.595,A -85,B 0,C 180,E1 -22082.588,E2 -22082.588} C_VEL
LIN {X 0,Y 203.32,Z 490.627,A -85,B 0,C 180,E1 -22085.379,E2 -22085.379} C_VEL
LIN {X 0,Y 207.718,Z 479.783,A -85,B 0,C 180,E1 -22087.825,E2 -22087.825} C_VEL
LIN {X 0,Y 212.615,Z 466.732,A -85,B 0,C 180,E1 -22090.134,E2 -22090.134} C_VEL
LIN {X 0,Y 216.699,Z 453.657,A -85,B 0,C 180,E1 -22091.982,E2 -22091.982} C_VEL
LIN {X 0,Y 220.144,Z 441.176,A -85,B 0,C 180,E1 -22093.344,E2 -22093.344} C_VEL
LIN {X 0,Y 223.426,Z 426.477,A -85,B 0,C 180,E1 -22094.576,E2 -22094.576} C_VEL
LIN {X 0,Y 225.967,Z 411.918,A -85,B 0,C 180,E1 -22095.433,E2 -22095.433} C_VEL
LIN {X 0,Y 227.595,Z 396.983,A -85,B 0,C 180,E1 -22096.044,E2 -22096.044} C_VEL
LIN {X 0,Y 233.193,Z 312.228,A -85,B 0,C 180,E1 -22098.468,E2 -22098.468} C_VEL
LIN {X 0,Y 227.516,Z 299.554,A -85,B 0,C 180,E1 -22100.639,E2 -22100.639} C_VEL
LIN {X 0,Y 222.462,Z 289.636,A -85,B 0,C 180,E1 -22102.681,E2 -22102.681} C_VEL
LIN {X 0,Y 216.696,Z 279.448,A -85,B 0,C 180,E1 -22105.187,E2 -22105.187} C_VEL
LIN {X 0,Y 211.59,Z 271.152,A -85,B 0,C 180,E1 -22107.616,E2 -22107.616} C_VEL
LIN {X 0,Y 205.921,Z 262.568,A -85,B 0,C 180,E1 -22110.619,E2 -22110.619} C_VEL
LIN {X 0,Y 201.406,Z 256.401,A -85,B 0,C 180,E1 -22113.304,E2 -22113.304} C_VEL
LIN {X 0,Y 197.851,Z 251.635,A -85,B 0,C 180,E1 -22115.681,E2 -22115.681} C_VEL
LIN {X 0,Y 192.387,Z 244.77,A -85,B 0,C 180,E1 -22120.112,E2 -22120.112} C_VEL
LIN {X 0,Y 190.921,Z 240.926,A -85,B 0,C 180,E1 -22125.068,E2 -22125.068} C_VEL
LIN {X 0,Y 189.661,Z 237.563,A -85,B 0,C 180,E1 -22131.476,E2 -22131.476} C_VEL
LIN {X 0,Y 189.433,Z 236.755,A -85,B 0,C 180,E1 -22133.61,E2 -22133.61} C_VEL
LIN {X 0,Y 189.108,Z 235.492,A -85,B 0,C 180,E1 -22140,E2 -22140} C_VEL
LIN {X 0,Y 189.134,Z 236.289,A -85,B 0,C 180,E1 -22147.122,E2 -22147.122} C_VEL
LIN {X 0,Y 189.345,Z 236.564,A -85,B 0,C 180,E1 -22148.539,E2 -22148.539} C_VEL
LIN {X 0,Y 189.675,Z 238.331,A -85,B 0,C 180,E1 -22152.846,E2 -22152.846} C_VEL
LIN {X 0,Y 190.629,Z 240.515,A -85,B 0,C 180,E1 -22157.154,E2 -22157.154} C_VEL
LIN {X 0,Y 192.311,Z 244.701,A -85,B 0,C 180,E1 -22162.817,E2 -22162.817} C_VEL
LIN {X 0,Y 197.923,Z 252.039,A -85,B 0,C 180,E1 -22167.357,E2 -22167.357} C_VEL
LIN {X 0,Y 202.313,Z 257.784,A -85,B 0,C 180,E1 -22170.225,E2 -22170.225} C_VEL
LIN {X 0,Y 206.561,Z 263.77,A -85,B 0,C 180,E1 -22172.692,E2 -22172.692} C_VEL
LIN {X 0,Y 210.117,Z 269.106,A -85,B 0,C 180,E1 -22174.581,E2 -22174.581} C_VEL
LIN {X 0,Y 215.71,Z 277.877,A -85,B 0,C 180,E1 -22177.276,E2 -22177.276} C_VEL
LIN {X 0,Y 222.302,Z 289.561,A -85,B 0,C 180,E1 -22180.15,E2 -22180.15} C_VEL
LIN {X 0,Y 228.678,Z 302.387,A -85,B 0,C 180,E1 -22182.684,E2 -22182.684} C_VEL
LIN {X 0,Y 232.948,Z 312.147,A -85,B 0,C 180,E1 -22184.289,E2 -22184.289} C_VEL
LIN {X 0,Y 227.917,Z 393.556,A -85,B 0,C 180,E1 -22186.527,E2 -22186.527} C_VEL
LIN {X 0,Y 226.136,Z 408.365,A -85,B 0,C 180,E1 -22187.244,E2 -22187.244} C_VEL
LIN {X 0,Y 223.869,Z 421.41,A -85,B 0,C 180,E1 -22188.155,E2 -22188.155} C_VEL
LIN {X 0,Y 220.991,Z 433.977,A -85,B 0,C 180,E1 -22189.311,E2 -22189.311} C_VEL
LIN {X 0,Y 217.514,Z 446.494,A -85,B 0,C 180,E1 -22190.809,E2 -22190.809} C_VEL
LIN {X 0,Y 213.488,Z 459.128,A -85,B 0,C 180,E1 -22192.778,E2 -22192.778} C_VEL
LIN {X 0,Y 209.638,Z 469.106,A -85,B 0,C 180,E1 -22194.669,E2 -22194.669} C_VEL
LIN {X 0,Y 205.007,Z 480.21,A -85,B 0,C 180,E1 -22197.32,E2 -22197.32} C_VEL
LIN {X 0,Y 200.749,Z 489.404,A -85,B 0,C 180,E1 -22200.074,E2 -22200.074} C_VEL
LIN {X 0,Y 196.487,Z 497.971,A -85,B 0,C 180,E1 -22203.295,E2 -22203.295} C_VEL
LIN {X 0,Y 193.362,Z 504.504,A -85,B 0,C 180,E1 -22206.433,E2 -22206.433} C_VEL
LIN {X 0,Y 189.551,Z 511.321,A -85,B 0,C 180,E1 -22210.506,E2 -22210.506} C_VEL
LIN {X 0,Y 186.916,Z 516.505,A -85,B 0,C 180,E1 -22214.739,E2 -22214.739} C_VEL
LIN {X 0,Y 185.076,Z 520.26,A -85,B 0,C 180,E1 -22219.054,E2 -22219.054} C_VEL
LIN {X 0,Y 184.01,Z 522.712,A -85,B 0,C 180,E1 -22223.42,E2 -22223.42} C_VEL
LIN {X 0,Y 183.507,Z 523.934,A -85,B 0,C 180,E1 -22227.804,E2 -22227.804} C_VEL
LIN {X 0,Y 183.497,Z 523.953,A -85,B 0,C 180,E1 -22232.194,E2 -22232.194} C_VEL
LIN {X 0,Y 183.941,Z 522.775,A -85,B 0,C 180,E1 -22236.581,E2 -22236.581} C_VEL
LIN {X 0,Y 184.996,Z 520.367,A -85,B 0,C 180,E1 -22240.949,E2 -22240.949} C_VEL
LIN {X 0,Y 186.858,Z 516.651,A -85,B 0,C 180,E1 -22245.264,E2 -22245.264} C_VEL
LIN {X 0,Y 189.478,Z 511.532,A -85,B 0,C 180,E1 -22249.5,E2 -22249.5} C_VEL
LIN {X 0,Y 192.221,Z 506.612,A -85,B 0,C 180,E1 -22252.574,E2 -22252.574} C_VEL
LIN {X 0,Y 195.824,Z 499.428,A -85,B 0,C 180,E1 -22256.202,E2 -22256.202} C_VEL
LIN {X 0,Y 199.956,Z 491.125,A -85,B 0,C 180,E1 -22259.475,E2 -22259.475} C_VEL
LIN {X 0,Y 204.204,Z 482.265,A -85,B 0,C 180,E1 -22262.238,E2 -22262.238} C_VEL
LIN {X 0,Y 208.723,Z 471.623,A -85,B 0,C 180,E1 -22264.917,E2 -22264.917} C_VEL
LIN {X 0,Y 212.936,Z 460.926,A -85,B 0,C 180,E1 -22267.037,E2 -22267.037} C_VEL
LIN {X 0,Y 216.844,Z 449.172,A -85,B 0,C 180,E1 -22268.935,E2 -22268.935} C_VEL
LIN {X 0,Y 220.402,Z 436.72,A -85,B 0,C 180,E1 -22270.517,E2 -22270.517} C_VEL
LIN {X 0,Y 223.704,Z 422.648,A -85,B 0,C 180,E1 -22271.881,E2 -22271.881} C_VEL
LIN {X 0,Y 226.267,Z 408.499,A -85,B 0,C 180,E1 -22272.875,E2 -22272.875} C_VEL
LIN {X 0,Y 228.013,Z 394.182,A -85,B 0,C 180,E1 -22273.574,E2 -22273.574} C_VEL
LIN {X 0,Y 230.553,Z 355.42,A -85,B 0,C 180,E1 -22274.655,E2 -22274.655} C_VEL
LIN {X 0,Y 233.024,Z 312.133,A -85,B 0,C 180,E1 -22275.858,E2 -22275.858} C_VEL
LIN {X 0,Y 227.738,Z 300.171,A -85,B 0,C 180,E1 -22277.861,E2 -22277.861} C_VEL
LIN {X 0,Y 221.69,Z 288.349,A -85,B 0,C 180,E1 -22280.297,E2 -22280.297} C_VEL
LIN {X 0,Y 216.133,Z 278.652,A -85,B 0,C 180,E1 -22282.725,E2 -22282.725} C_VEL
LIN {X 0,Y 211.599,Z 271.325,A -85,B 0,C 180,E1 -22284.889,E2 -22284.889} C_VEL
LIN {X 0,Y 208.222,Z 266.188,A -85,B 0,C 180,E1 -22286.631,E2 -22286.631} C_VEL
LIN {X 0,Y 205.081,Z 261.573,A -85,B 0,C 180,E1 -22288.377,E2 -22288.377} C_VEL
LIN {X 0,Y 201.035,Z 256.084,A -85,B 0,C 180,E1 -22290.826,E2 -22290.826} C_VEL
LIN {X 0,Y 196.546,Z 250.306,A -85,B 0,C 180,E1 -22293.91,E2 -22293.91} C_VEL
LIN {X 0,Y 192.198,Z 244.477,A -85,B 0,C 180,E1 -22297.716,E2 -22297.716} C_VEL
LIN {X 0,Y 190.639,Z 240.385,A -85,B 0,C 180,E1 -22303.43,E2 -22303.43} C_VEL
LIN {X 0,Y 189.578,Z 237.593,A -85,B 0,C 180,E1 -22309.318,E2 -22309.318} C_VEL
LIN {X 0,Y 189.468,Z 236.778,A -85,B 0,C 180,E1 -22311.467,E2 -22311.467} C_VEL
LIN {X 0,Y 189.097,Z 235.786,A -85,B 0,C 180,E1 -22317.87,E2 -22317.87} C_VEL
LIN {X 0,Y 189.247,Z 235.674,A -85,B 0,C 180,E1 -22320,E2 -22320} C_VEL
LIN {X 0,Y 189.242,Z 236.457,A -85,B 0,C 180,E1 -22324.259,E2 -22324.259} C_VEL
LIN {X 0,Y 189.547,Z 236.945,A -85,B 0,C 180,E1 -22326.386,E2 -22326.386} C_VEL
LIN {X 0,Y 190.037,Z 238.763,A -85,B 0,C 180,E1 -22330.656,E2 -22330.656} C_VEL
LIN {X 0,Y 191.005,Z 241.122,A -85,B 0,C 180,E1 -22334.925,E2 -22334.925} C_VEL
LIN {X 0,Y 192.431,Z 244.895,A -85,B 0,C 180,E1 -22339.744,E2 -22339.744} C_VEL
LIN {X 0,Y 198.232,Z 252.193,A -85,B 0,C 180,E1 -22344.409,E2 -22344.409} C_VEL
LIN {X 0,Y 202.827,Z 258.357,A -85,B 0,C 180,E1 -22347.424,E2 -22347.424} C_VEL
LIN {X 0,Y 207.087,Z 264.368,A -85,B 0,C 180,E1 -22349.898,E2 -22349.898} C_VEL
LIN {X 0,Y 211.993,Z 271.684,A -85,B 0,C 180,E1 -22352.455,E2 -22352.455} C_VEL
LIN {X 0,Y 218.179,Z 281.752,A -85,B 0,C 180,E1 -22355.361,E2 -22355.361} C_VEL
LIN {X 0,Y 225.261,Z 294.897,A -85,B 0,C 180,E1 -22358.371,E2 -22358.371} C_VEL
LIN {X 0,Y 230.733,Z 306.28,A -85,B 0,C 180,E1 -22360.514,E2 -22360.514} C_VEL
LIN {X 0,Y 231.231,Z 307.464,A -85,B 0,C 180,E1 -22360.706,E2 -22360.706} C_VEL
LIN {X 0,Y 231.781,Z 310.303,A -85,B 0,C 180,E1 -22360.988,E2 -22360.988} C_VEL
LIN {X 0,Y 231.491,Z 313.503,A -85,B 0,C 180,E1 -22361.057,E2 -22361.057} C_VEL
LIN {X 0,Y 230.501,Z 317.349,A -85,B 0,C 180,E1 -22360.966,E2 -22360.966} C_VEL
LIN {X 0,Y 227.93,Z 325.594,A -85,B 0,C 180,E1 -22360.645,E2 -22360.645} C_VEL
LIN {X 0,Y 227.513,Z 328.436,A -85,B 0,C 180,E1 -22360.664,E2 -22360.664} C_VEL
LIN {X 0,Y 222.389,Z 401.671,A -85,B 0,C 180,E1 -22362.799,E2 -22362.799} C_VEL
LIN {X 0,Y 220.216,Z 417.258,A -85,B 0,C 180,E1 -22363.529,E2 -22363.529} C_VEL
LIN {X 0,Y 217.414,Z 431.543,A -85,B 0,C 180,E1 -22364.508,E2 -22364.508} C_VEL
LIN {X 0,Y 214.016,Z 445.06,A -85,B 0,C 180,E1 -22365.749,E2 -22365.749} C_VEL
LIN {X 0,Y 210.18,Z 457.875,A -85,B 0,C 180,E1 -22367.286,E2 -22367.286} C_VEL
LIN {X 0,Y 205.84,Z 470.514,A -85,B 0,C 180,E1 -22369.235,E2 -22369.235} C_VEL
LIN {X 0,Y 200.879,Z 482.834,A -85,B 0,C 180,E1 -22371.612,E2 -22371.612} C_VEL
LIN {X 0,Y 195.961,Z 494.01,A -85,B 0,C 180,E1 -22374.354,E2 -22374.354} C_VEL
LIN {X 0,Y 191.228,Z 504.251,A -85,B 0,C 180,E1 -22377.551,E2 -22377.551} C_VEL
LIN {X 0,Y 186.773,Z 513.725,A -85,B 0,C 180,E1 -22381.331,E2 -22381.331} C_VEL
LIN {X 0,Y 183.079,Z 521.089,A -85,B 0,C 180,E1 -22385.024,E2 -22385.024} C_VEL
LIN {X 0,Y 179.919,Z 527.866,A -85,B 0,C 180,E1 -22389.419,E2 -22389.419} C_VEL
LIN {X 0,Y 177.757,Z 533.117,A -85,B 0,C 180,E1 -22393.934,E2 -22393.934} C_VEL
LIN {X 0,Y 176.45,Z 536.974,A -85,B 0,C 180,E1 -22398.514,E2 -22398.514} C_VEL
LIN {X 0,Y 176.103,Z 539.526,A -85,B 0,C 180,E1 -22403.125,E2 -22403.125} C_VEL
LIN {X 0,Y 176.144,Z 540.439,A -85,B 0,C 180,E1 -22405.926,E2 -22405.926} C_VEL
LIN {X 0,Y 176.326,Z 540.975,A -85,B 0,C 180,E1 -22410.001,E2 -22410.001} C_VEL
LIN {X 0,Y 176.122,Z 540.309,A -85,B 0,C 180,E1 -22414.578,E2 -22414.578} C_VEL
LIN {X 0,Y 176.189,Z 538.371,A -85,B 0,C 180,E1 -22419.182,E2 -22419.182} C_VEL
LIN {X 0,Y 176.968,Z 535.156,A -85,B 0,C 180,E1 -22423.786,E2 -22423.786} C_VEL
LIN {X 0,Y 178.763,Z 530.602,A -85,B 0,C 180,E1 -22428.332,E2 -22428.332} C_VEL
LIN {X 0,Y 181.39,Z 524.579,A -85,B 0,C 180,E1 -22432.797,E2 -22432.797} C_VEL
LIN {X 0,Y 185.044,Z 516.936,A -85,B 0,C 180,E1 -22437.114,E2 -22437.114} C_VEL
LIN {X 0,Y 189.092,Z 508.691,A -85,B 0,C 180,E1 -22440.734,E2 -22440.734} C_VEL
LIN {X 0,Y 193.695,Z 498.722,A -85,B 0,C 180,E1 -22444.222,E2 -22444.222} C_VEL
LIN {X 0,Y 198.363,Z 488.449,A -85,B 0,C 180,E1 -22447.036,E2 -22447.036} C_VEL
LIN {X 0,Y 202.612,Z 478.316,A -85,B 0,C 180,E1 -22449.275,E2 -22449.275} C_VEL
LIN {X 0,Y 207.134,Z 466.445,A -85,B 0,C 180,E1 -22451.392,E2 -22451.392} C_VEL
LIN {X 0,Y 211.45,Z 453.207,A -85,B 0,C 180,E1 -22453.276,E2 -22453.276} C_VEL
LIN {X 0,Y 214.997,Z 440.67,A -85,B 0,C 180,E1 -22454.653,E2 -22454.653} C_VEL
LIN {X 0,Y 218.43,Z 425.888,A -85,B 0,C 180,E1 -22455.882,E2 -22455.882} C_VEL
LIN {X 0,Y 220.893,Z 412.075,A -85,B 0,C 180,E1 -22456.702,E2 -22456.702} C_VEL
LIN {X 0,Y 222.578,Z 397.436,A -85,B 0,C 180,E1 -22457.312,E2 -22457.312} C_VEL
LIN {X 0,Y 228.228,Z 314.657,A -85,B 0,C 180,E1 -22459.709,E2 -22459.709} C_VEL
LIN {X 0,Y 222.924,Z 302.708,A -85,B 0,C 180,E1 -22461.865,E2 -22461.865} C_VEL
LIN {X 0,Y 216.697,Z 290.513,A -85,B 0,C 180,E1 -22464.572,E2 -22464.572} C_VEL
LIN {X 0,Y 211.385,Z 281.306,A -85,B 0,C 180,E1 -22467.086,E2 -22467.086} C_VEL
LIN {X 0,Y 207.703,Z 275.305,A -85,B 0,C 180,E1 -22468.982,E2 -22468.982} C_VEL
LIN {X 0,Y 202.4,Z 267.292,A -85,B 0,C 180,E1 -22471.992,E2 -22471.992} C_VEL
LIN {X 0,Y 198.905,Z 262.328,A -85,B 0,C 180,E1 -22474.212,E2 -22474.212} C_VEL
LIN {X 0,Y 194.962,Z 257.006,A -85,B 0,C 180,E1 -22477.018,E2 -22477.018} C_VEL
LIN {X 0,Y 189.825,Z 250.571,A -85,B 0,C 180,E1 -22481.378,E2 -22481.378} C_VEL
LIN {X 0,Y 185.232,Z 244.748,A -85,B 0,C 180,E1 -22486.772,E2 -22486.772} C_VEL
LIN {X 0,Y 184.249,Z 241.904,A -85,B 0,C 180,E1 -22492.633,E2 -22492.633} C_VEL
LIN {X 0,Y 183.844,Z 240.592,A -85,B 0,C 180,E1 -22497.81,E2 -22497.81} C_VEL
LIN {X 0,Y 183.879,Z 240.274,A -85,B 0,C 180,E1 -22500,E2 -22500} C_VEL
LIN {X 0,Y 183.872,Z 241.064,A -85,B 0,C 180,E1 -22507.165,E2 -22507.165} C_VEL
LIN {X 0,Y 184.085,Z 241.403,A -85,B 0,C 180,E1 -22508.785,E2 -22508.785} C_VEL
LIN {X 0,Y 185.032,Z 244.507,A -85,B 0,C 180,E1 -22515.798,E2 -22515.798} C_VEL
LIN {X 0,Y 186.085,Z 246.264,A -85,B 0,C 180,E1 -22517.587,E2 -22517.587} C_VEL
LIN {X 0,Y 190.87,Z 251.834,A -85,B 0,C 180,E1 -22522.554,E2 -22522.554} C_VEL
LIN {X 0,Y 195.96,Z 258.492,A -85,B 0,C 180,E1 -22526.69,E2 -22526.69} C_VEL
LIN {X 0,Y 200.02,Z 263.985,A -85,B 0,C 180,E1 -22529.467,E2 -22529.467} C_VEL
LIN {X 0,Y 204.011,Z 269.762,A -85,B 0,C 180,E1 -22531.895,E2 -22531.895} C_VEL
LIN {X 0,Y 207.292,Z 274.827,A -85,B 0,C 180,E1 -22533.723,E2 -22533.723} C_VEL
LIN {X 0,Y 212.418,Z 283.063,A -85,B 0,C 180,E1 -22536.323,E2 -22536.323} C_VEL
LIN {X 0,Y 218.871,Z 294.851,A -85,B 0,C 180,E1 -22539.285,E2 -22539.285} C_VEL
LIN {X 0,Y 224.943,Z 307.418,A -85,B 0,C 180,E1 -22541.824,E2 -22541.824} C_VEL
LIN {X 0,Y 228.05,Z 314.697,A -85,B 0,C 180,E1 -22543.061,E2 -22543.061} C_VEL
LIN {X 0,Y 222.932,Z 393.665,A -85,B 0,C 180,E1 -22545.245,E2 -22545.245} C_VEL
LIN {X 0,Y 221.123,Z 408.264,A -85,B 0,C 180,E1 -22545.952,E2 -22545.952} C_VEL
